// Mitsubishi GX Works2 project: BAJAJ-N5K-Q CONV-18.08.22_MOD2   PLC: Q03UDV

PROGRAM MAIN
0     END
END_PROGRAM

PROGRAM 1_ALARMS  // ALL
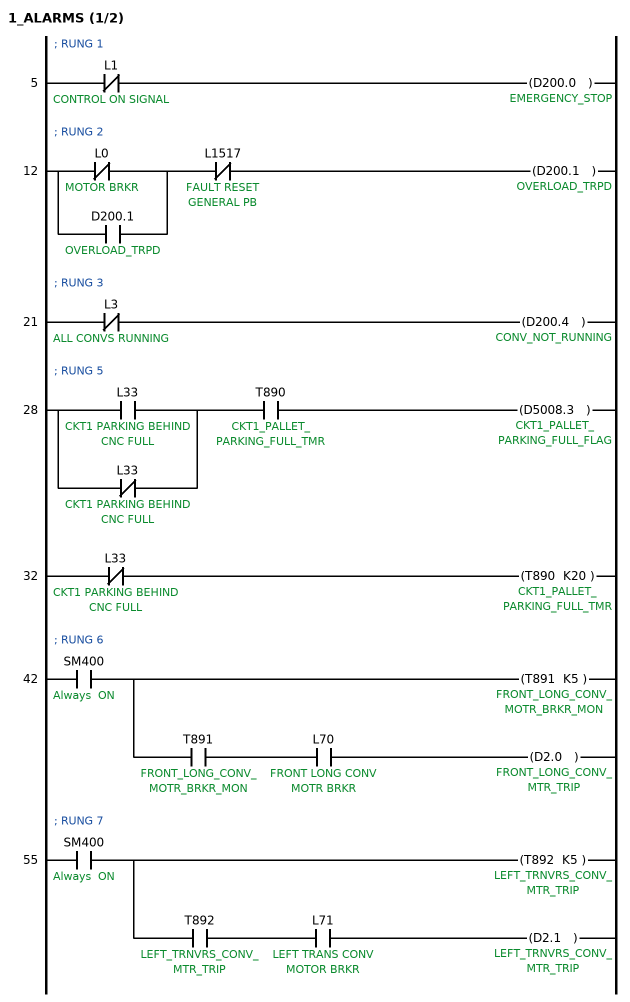
; RUNG 1
5     LDI     L1  ; CONTROL ON SIGNAL
      OUT     D200.0  ; EMERGENCY_STOP
; RUNG 2
12    LDI     L0  ; MOTOR BRKR
      OR      D200.1  ; OVERLOAD_TRPD
      ANI     L1517  ; FAULT RESET GENERAL PB
      OUT     D200.1  ; OVERLOAD_TRPD
; RUNG 3
21    LDI     L3  ; ALL CONVS RUNNING
      OUT     D200.4  ; CONV_NOT_RUNNING
; RUNG 5
28    LD      L33  ; CKT1 PARKING BEHIND CNC FULL
      ORI     L33  ; CKT1 PARKING BEHIND CNC FULL
      AND     T890  ; CKT1_PALLET_PARKING_FULL_TMR
      OUT     D5008.3  ; CKT1_PALLET_PARKING_FULL_FLAG
32    LDI     L33  ; CKT1 PARKING BEHIND CNC FULL
      OUT     T890 K20  ; CKT1_PALLET_PARKING_FULL_TMR
; RUNG 6
42    LD      SM400  ; Always  ON
      OUT     T891 K5  ; FRONT_LONG_CONV_MOTR_BRKR_MON
      AND     T891  ; FRONT_LONG_CONV_MOTR_BRKR_MON
      AND     L70  ; FRONT LONG CONV MOTR BRKR
      OUT     D2.0  ; FRONT_LONG_CONV_MTR_TRIP
; RUNG 7
55    LD      SM400  ; Always  ON
      OUT     T892 K5  ; LEFT_TRNVRS_CONV_MTR_TRIP
      AND     T892  ; LEFT_TRNVRS_CONV_MTR_TRIP
      AND     L71  ; LEFT TRANS CONV MOTOR BRKR
      OUT     D2.1  ; LEFT_TRNVRS_CONV_MTR_TRIP
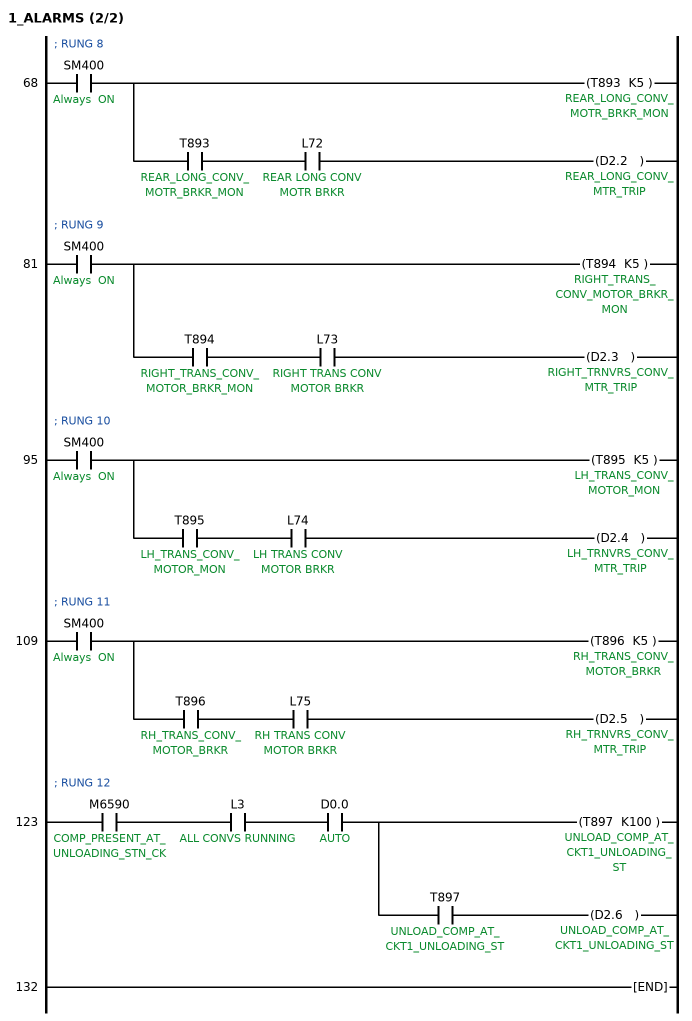
; RUNG 8
68    LD      SM400  ; Always  ON
      OUT     T893 K5  ; REAR_LONG_CONV_MOTR_BRKR_MON
      AND     T893  ; REAR_LONG_CONV_MOTR_BRKR_MON
      AND     L72  ; REAR LONG CONV MOTR BRKR
      OUT     D2.2  ; REAR_LONG_CONV_MTR_TRIP
; RUNG 9
81    LD      SM400  ; Always  ON
      OUT     T894 K5  ; RIGHT_TRANS_CONV_MOTOR_BRKR_MON
      AND     T894  ; RIGHT_TRANS_CONV_MOTOR_BRKR_MON
      AND     L73  ; RIGHT TRANS CONV MOTOR BRKR
      OUT     D2.3  ; RIGHT_TRNVRS_CONV_MTR_TRIP
; RUNG 10
95    LD      SM400  ; Always  ON
      OUT     T895 K5  ; LH_TRANS_CONV_MOTOR_MON
      AND     T895  ; LH_TRANS_CONV_MOTOR_MON
      AND     L74  ; LH TRANS CONV MOTOR BRKR
      OUT     D2.4  ; LH_TRNVRS_CONV_MTR_TRIP
; RUNG 11
109   LD      SM400  ; Always  ON
      OUT     T896 K5  ; RH_TRANS_CONV_MOTOR_BRKR
      AND     T896  ; RH_TRANS_CONV_MOTOR_BRKR
      AND     L75  ; RH TRANS CONV MOTOR BRKR
      OUT     D2.5  ; RH_TRNVRS_CONV_MTR_TRIP
; RUNG 12
123   LD      M6590  ; COMP_PRESENT_AT_UNLOADING_STN_CK
      AND     L3  ; ALL CONVS RUNNING
      AND     D0.0  ; AUTO
      OUT     T897 K100  ; UNLOAD_COMP_AT_CKT1_UNLOADING_ST
      AND     T897  ; UNLOAD_COMP_AT_CKT1_UNLOADING_ST
      OUT     D2.6  ; UNLOAD_COMP_AT_CKT1_UNLOADING_ST
132   END
END_PROGRAM

PROGRAM 2_AUTO  // UNLOADER
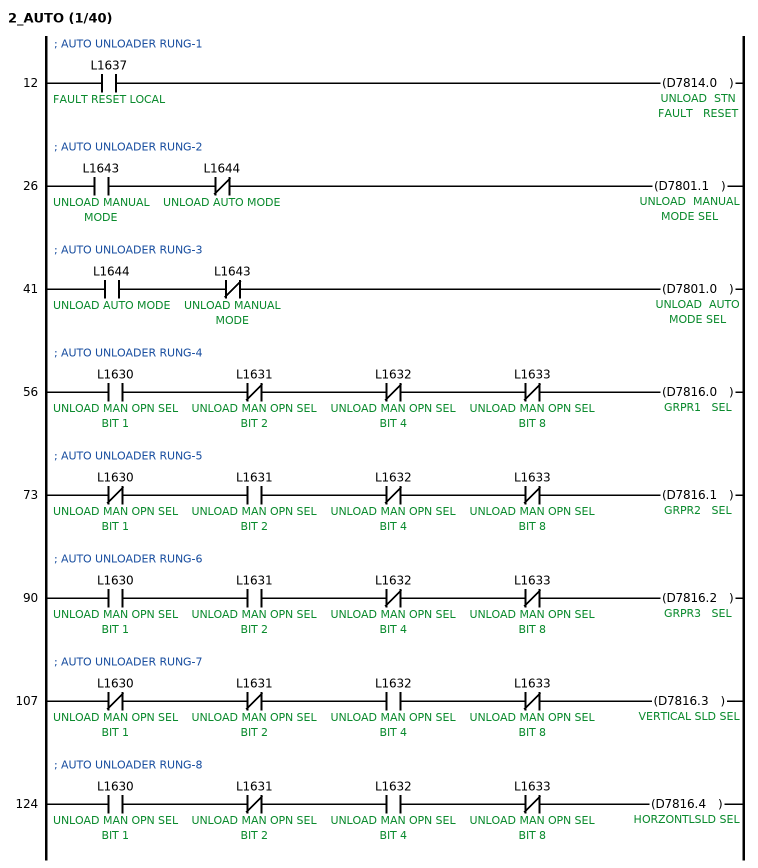
; AUTO UNLOADER RUNG-1
12    LD      L1637  ; FAULT RESET LOCAL
      OUT     D7814.0  ; UNLOAD  STN     FAULT   RESET
; AUTO UNLOADER RUNG-2
26    LD      L1643  ; UNLOAD MANUAL MODE
      ANI     L1644  ; UNLOAD AUTO MODE
      OUT     D7801.1  ; UNLOAD  MANUAL  MODE SEL
; AUTO UNLOADER RUNG-3
41    LD      L1644  ; UNLOAD AUTO MODE
      ANI     L1643  ; UNLOAD MANUAL MODE
      OUT     D7801.0  ; UNLOAD  AUTO    MODE SEL
; AUTO UNLOADER RUNG-4
56    LD      L1630  ; UNLOAD MAN OPN SEL BIT 1
      ANI     L1631  ; UNLOAD MAN OPN SEL BIT 2
      ANI     L1632  ; UNLOAD MAN OPN SEL BIT 4
      ANI     L1633  ; UNLOAD MAN OPN SEL BIT 8
      OUT     D7816.0  ; GRPR1   SEL
; AUTO UNLOADER RUNG-5
73    LDI     L1630  ; UNLOAD MAN OPN SEL BIT 1
      AND     L1631  ; UNLOAD MAN OPN SEL BIT 2
      ANI     L1632  ; UNLOAD MAN OPN SEL BIT 4
      ANI     L1633  ; UNLOAD MAN OPN SEL BIT 8
      OUT     D7816.1  ; GRPR2   SEL
; AUTO UNLOADER RUNG-6
90    LD      L1630  ; UNLOAD MAN OPN SEL BIT 1
      AND     L1631  ; UNLOAD MAN OPN SEL BIT 2
      ANI     L1632  ; UNLOAD MAN OPN SEL BIT 4
      ANI     L1633  ; UNLOAD MAN OPN SEL BIT 8
      OUT     D7816.2  ; GRPR3   SEL
; AUTO UNLOADER RUNG-7
107   LDI     L1630  ; UNLOAD MAN OPN SEL BIT 1
      ANI     L1631  ; UNLOAD MAN OPN SEL BIT 2
      AND     L1632  ; UNLOAD MAN OPN SEL BIT 4
      ANI     L1633  ; UNLOAD MAN OPN SEL BIT 8
      OUT     D7816.3  ; VERTICAL SLD SEL
; AUTO UNLOADER RUNG-8
124   LD      L1630  ; UNLOAD MAN OPN SEL BIT 1
      ANI     L1631  ; UNLOAD MAN OPN SEL BIT 2
      AND     L1632  ; UNLOAD MAN OPN SEL BIT 4
      ANI     L1633  ; UNLOAD MAN OPN SEL BIT 8
      OUT     D7816.4  ; HORZONTLSLD SEL
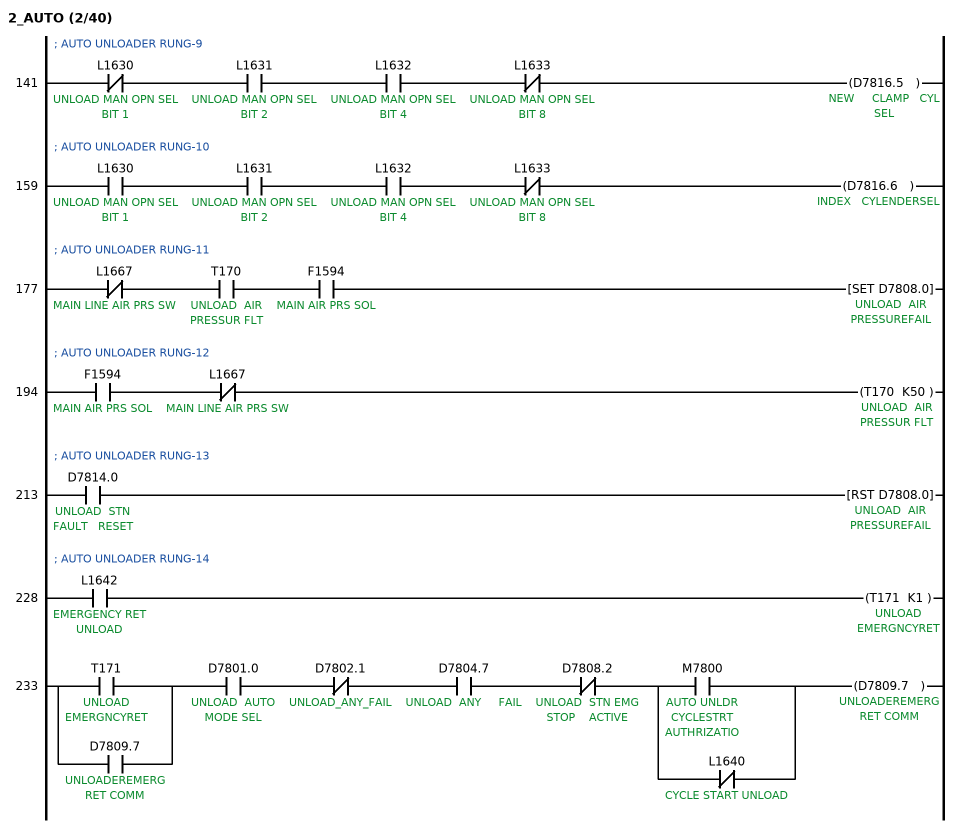
; AUTO UNLOADER RUNG-9
141   LDI     L1630  ; UNLOAD MAN OPN SEL BIT 1
      AND     L1631  ; UNLOAD MAN OPN SEL BIT 2
      AND     L1632  ; UNLOAD MAN OPN SEL BIT 4
      ANI     L1633  ; UNLOAD MAN OPN SEL BIT 8
      OUT     D7816.5  ; NEW     CLAMP   CYL SEL
; AUTO UNLOADER RUNG-10
159   LD      L1630  ; UNLOAD MAN OPN SEL BIT 1
      AND     L1631  ; UNLOAD MAN OPN SEL BIT 2
      AND     L1632  ; UNLOAD MAN OPN SEL BIT 4
      ANI     L1633  ; UNLOAD MAN OPN SEL BIT 8
      OUT     D7816.6  ; INDEX   CYLENDERSEL
; AUTO UNLOADER RUNG-11
177   LDI     L1667  ; MAIN LINE AIR PRS SW
      AND     T170  ; UNLOAD  AIR     PRESSUR FLT
      AND     F1594  ; MAIN AIR PRS SOL
      SET     D7808.0  ; UNLOAD  AIR     PRESSUREFAIL
; AUTO UNLOADER RUNG-12
194   LD      F1594  ; MAIN AIR PRS SOL
      ANI     L1667  ; MAIN LINE AIR PRS SW
      OUT     T170 K50  ; UNLOAD  AIR     PRESSUR FLT
; AUTO UNLOADER RUNG-13
213   LD      D7814.0  ; UNLOAD  STN     FAULT   RESET
      RST     D7808.0  ; UNLOAD  AIR     PRESSUREFAIL
; AUTO UNLOADER RUNG-14
228   LD      L1642  ; EMERGENCY RET UNLOAD
      OUT     T171 K1  ; UNLOAD  EMERGNCYRET
233   LD      T171  ; UNLOAD  EMERGNCYRET
      OR      D7809.7  ; UNLOADEREMERG   RET COMM
      AND     D7801.0  ; UNLOAD  AUTO    MODE SEL
      ANI     D7802.1  ; UNLOAD_ANY_FAIL
      AND     D7804.7  ; UNLOAD  ANY     FAIL
      ANI     D7808.2  ; UNLOAD  STN EMG STOP    ACTIVE
      LD      M7800  ; AUTO UNLDR CYCLESTRT AUTHRIZATIO
      ORI     L1640  ; CYCLE START UNLOAD
      ANB
      OUT     D7809.7  ; UNLOADEREMERG   RET COMM
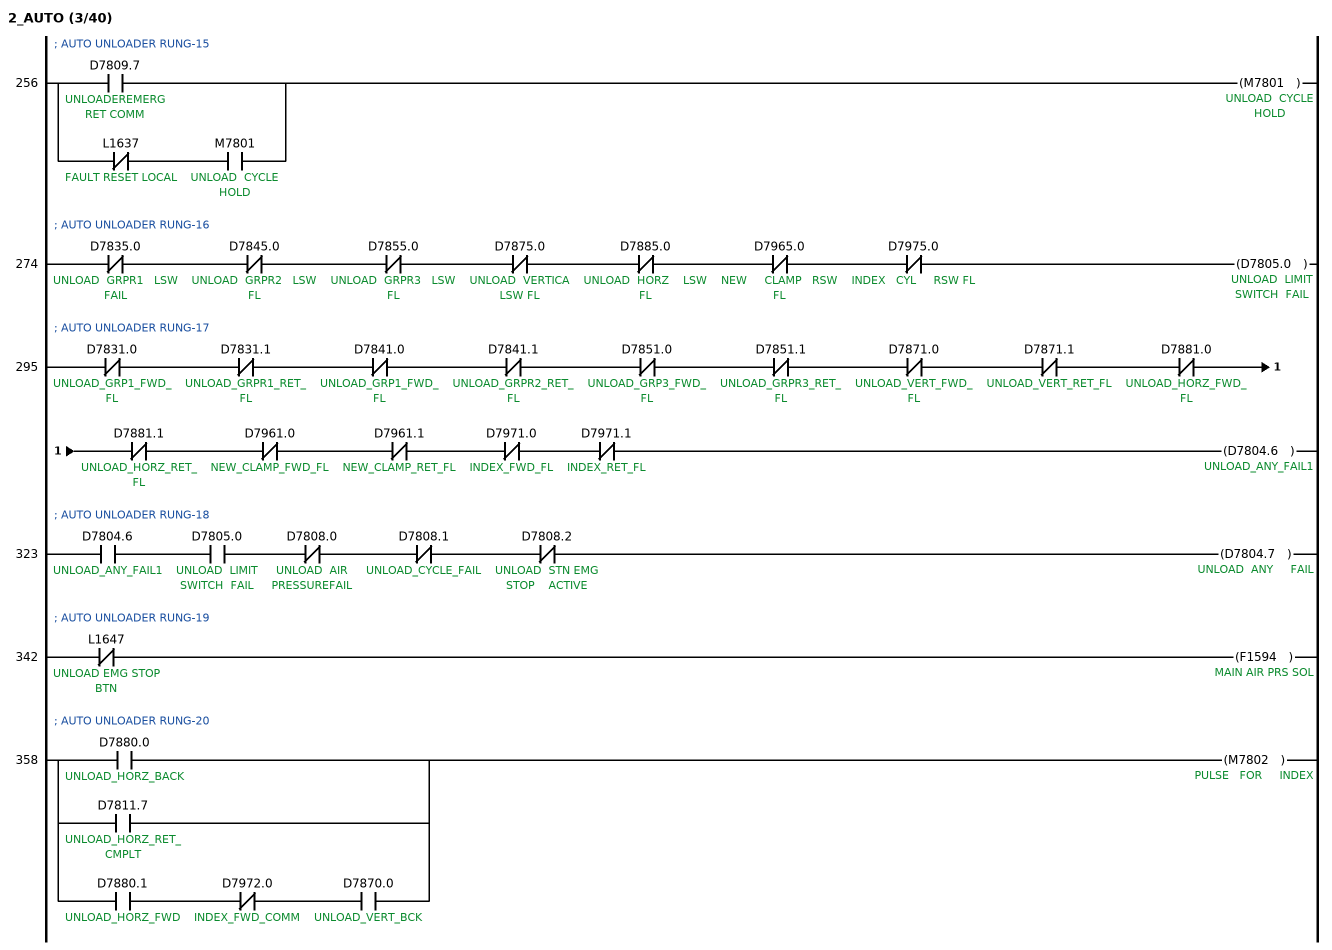
; AUTO UNLOADER RUNG-15
256   LD      D7809.7  ; UNLOADEREMERG   RET COMM
      LDI     L1637  ; FAULT RESET LOCAL
      AND     M7801  ; UNLOAD  CYCLE   HOLD
      ORB
      OUT     M7801  ; UNLOAD  CYCLE   HOLD
; AUTO UNLOADER RUNG-16
274   LDI     D7835.0  ; UNLOAD  GRPR1   LSW FAIL
      ANI     D7845.0  ; UNLOAD  GRPR2   LSW FL
      ANI     D7855.0  ; UNLOAD  GRPR3   LSW FL
      ANI     D7875.0  ; UNLOAD  VERTICA LSW FL
      ANI     D7885.0  ; UNLOAD  HORZ    LSW FL
      ANI     D7965.0  ; NEW     CLAMP   RSW FL
      ANI     D7975.0  ; INDEX   CYL     RSW FL
      OUT     D7805.0  ; UNLOAD  LIMIT   SWITCH  FAIL
; AUTO UNLOADER RUNG-17
295   LDI     D7831.0  ; UNLOAD_GRP1_FWD_FL
      ANI     D7831.1  ; UNLOAD_GRPR1_RET_FL
      ANI     D7841.0  ; UNLOAD_GRP1_FWD_FL
      ANI     D7841.1  ; UNLOAD_GRPR2_RET_FL
      ANI     D7851.0  ; UNLOAD_GRP3_FWD_FL
      ANI     D7851.1  ; UNLOAD_GRPR3_RET_FL
      ANI     D7871.0  ; UNLOAD_VERT_FWD_FL
      ANI     D7871.1  ; UNLOAD_VERT_RET_FL
      ANI     D7881.0  ; UNLOAD_HORZ_FWD_FL
      ANI     D7881.1  ; UNLOAD_HORZ_RET_FL
      ANI     D7961.0  ; NEW_CLAMP_FWD_FL
      ANI     D7961.1  ; NEW_CLAMP_RET_FL
      ANI     D7971.0  ; INDEX_FWD_FL
      ANI     D7971.1  ; INDEX_RET_FL
      OUT     D7804.6  ; UNLOAD_ANY_FAIL1
; AUTO UNLOADER RUNG-18
323   LD      D7804.6  ; UNLOAD_ANY_FAIL1
      AND     D7805.0  ; UNLOAD  LIMIT   SWITCH  FAIL
      ANI     D7808.0  ; UNLOAD  AIR     PRESSUREFAIL
      ANI     D7808.1  ; UNLOAD_CYCLE_FAIL
      ANI     D7808.2  ; UNLOAD  STN EMG STOP    ACTIVE
      OUT     D7804.7  ; UNLOAD  ANY     FAIL
; AUTO UNLOADER RUNG-19
342   LDI     L1647  ; UNLOAD EMG STOP BTN
      OUT     F1594  ; MAIN AIR PRS SOL
; AUTO UNLOADER RUNG-20
358   LD      D7880.0  ; UNLOAD_HORZ_BACK
      OR      D7811.7  ; UNLOAD_HORZ_RET_CMPLT
      LD      D7880.1  ; UNLOAD_HORZ_FWD
      ANI     D7972.0  ; INDEX_FWD_COMM
      AND     D7870.0  ; UNLOAD_VERT_BCK
      ORB
      OUT     M7802  ; PULSE   FOR     INDEX
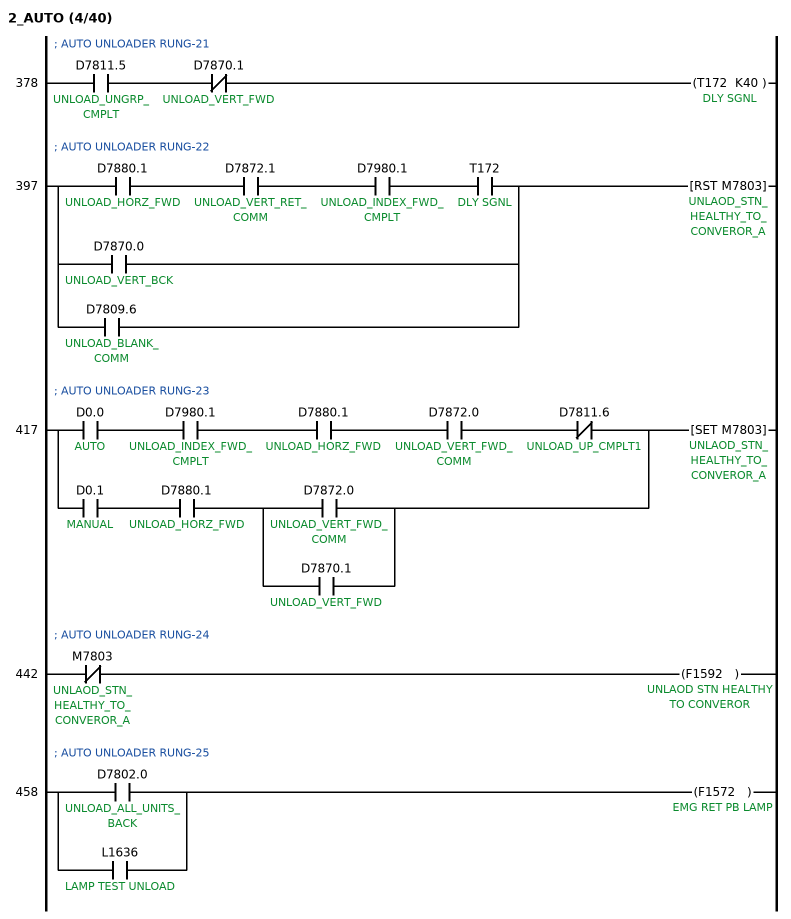
; AUTO UNLOADER RUNG-21
378   LD      D7811.5  ; UNLOAD_UNGRP_CMPLT
      ANI     D7870.1  ; UNLOAD_VERT_FWD
      OUT     T172 K40  ; DLY SGNL
; AUTO UNLOADER RUNG-22
397   LD      D7880.1  ; UNLOAD_HORZ_FWD
      AND     D7872.1  ; UNLOAD_VERT_RET_COMM
      AND     D7980.1  ; UNLOAD_INDEX_FWD_CMPLT
      AND     T172  ; DLY SGNL
      OR      D7870.0  ; UNLOAD_VERT_BCK
      OR      D7809.6  ; UNLOAD_BLANK_COMM
      RST     M7803  ; UNLAOD_STN_HEALTHY_TO_CONVEROR_A
; AUTO UNLOADER RUNG-23
417   LD      D0.0  ; AUTO
      AND     D7980.1  ; UNLOAD_INDEX_FWD_CMPLT
      AND     D7880.1  ; UNLOAD_HORZ_FWD
      AND     D7872.0  ; UNLOAD_VERT_FWD_COMM
      ANI     D7811.6  ; UNLOAD_UP_CMPLT1
      LD      D0.1  ; MANUAL
      AND     D7880.1  ; UNLOAD_HORZ_FWD
      LD      D7872.0  ; UNLOAD_VERT_FWD_COMM
      OR      D7870.1  ; UNLOAD_VERT_FWD
      ANB
      ORB
      SET     M7803  ; UNLAOD_STN_HEALTHY_TO_CONVEROR_A
; AUTO UNLOADER RUNG-24
442   LDI     M7803  ; UNLAOD_STN_HEALTHY_TO_CONVEROR_A
      OUT     F1592  ; UNLAOD STN HEALTHY TO CONVEROR
; AUTO UNLOADER RUNG-25
458   LD      D7802.0  ; UNLOAD_ALL_UNITS_BACK
      OR      L1636  ; LAMP TEST UNLOAD
      OUT     F1572  ; EMG RET PB LAMP
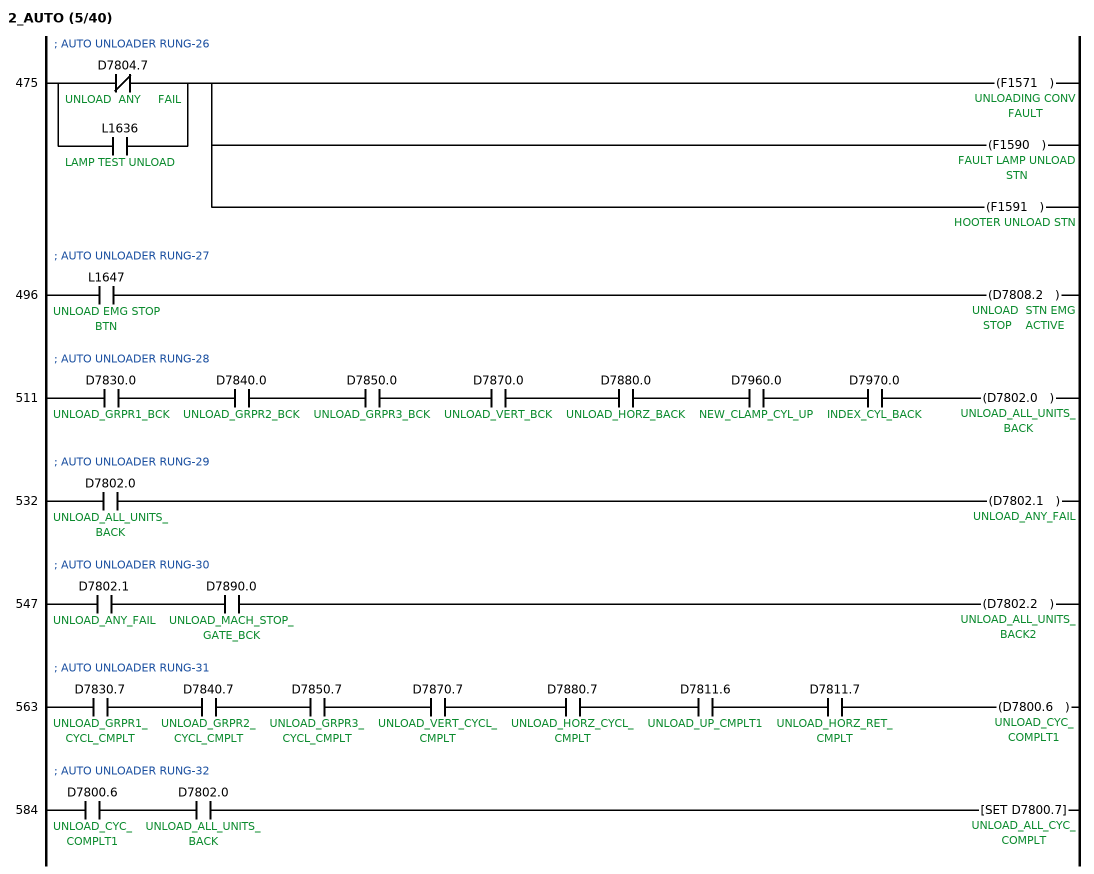
; AUTO UNLOADER RUNG-26
475   LDI     D7804.7  ; UNLOAD  ANY     FAIL
      OR      L1636  ; LAMP TEST UNLOAD
      OUT     F1571  ; UNLOADING CONV FAULT
      OUT     F1590  ; FAULT LAMP UNLOAD STN
      OUT     F1591  ; HOOTER UNLOAD STN
; AUTO UNLOADER RUNG-27
496   LD      L1647  ; UNLOAD EMG STOP BTN
      OUT     D7808.2  ; UNLOAD  STN EMG STOP    ACTIVE
; AUTO UNLOADER RUNG-28
511   LD      D7830.0  ; UNLOAD_GRPR1_BCK
      AND     D7840.0  ; UNLOAD_GRPR2_BCK
      AND     D7850.0  ; UNLOAD_GRPR3_BCK
      AND     D7870.0  ; UNLOAD_VERT_BCK
      AND     D7880.0  ; UNLOAD_HORZ_BACK
      AND     D7960.0  ; NEW_CLAMP_CYL_UP
      AND     D7970.0  ; INDEX_CYL_BACK
      OUT     D7802.0  ; UNLOAD_ALL_UNITS_BACK
; AUTO UNLOADER RUNG-29
532   LD      D7802.0  ; UNLOAD_ALL_UNITS_BACK
      OUT     D7802.1  ; UNLOAD_ANY_FAIL
; AUTO UNLOADER RUNG-30
547   LD      D7802.1  ; UNLOAD_ANY_FAIL
      AND     D7890.0  ; UNLOAD_MACH_STOP_GATE_BCK
      OUT     D7802.2  ; UNLOAD_ALL_UNITS_BACK2
; AUTO UNLOADER RUNG-31
563   LD      D7830.7  ; UNLOAD_GRPR1_CYCL_CMPLT
      AND     D7840.7  ; UNLOAD_GRPR2_CYCL_CMPLT
      AND     D7850.7  ; UNLOAD_GRPR3_CYCL_CMPLT
      AND     D7870.7  ; UNLOAD_VERT_CYCL_CMPLT
      AND     D7880.7  ; UNLOAD_HORZ_CYCL_CMPLT
      AND     D7811.6  ; UNLOAD_UP_CMPLT1
      AND     D7811.7  ; UNLOAD_HORZ_RET_CMPLT
      OUT     D7800.6  ; UNLOAD_CYC_COMPLT1
; AUTO UNLOADER RUNG-32
584   LD      D7800.6  ; UNLOAD_CYC_COMPLT1
      AND     D7802.0  ; UNLOAD_ALL_UNITS_BACK
      SET     D7800.7  ; UNLOAD_ALL_CYC_COMPLT
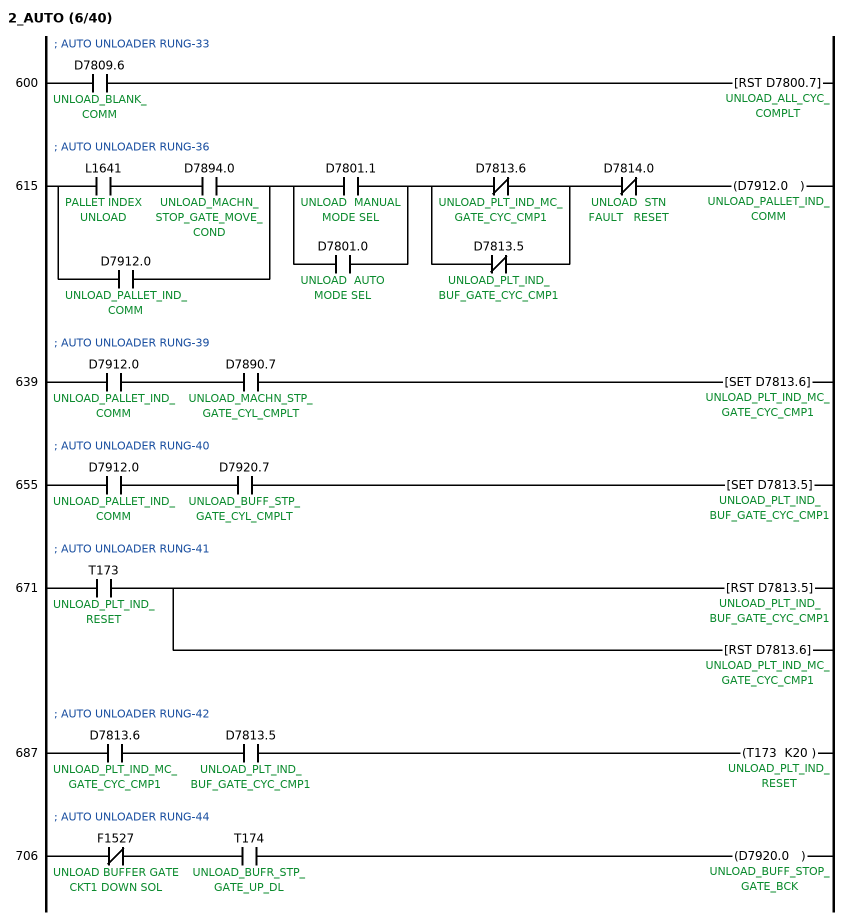
; AUTO UNLOADER RUNG-33
600   LD      D7809.6  ; UNLOAD_BLANK_COMM
      RST     D7800.7  ; UNLOAD_ALL_CYC_COMPLT
; AUTO UNLOADER RUNG-36
615   LD      L1641  ; PALLET INDEX UNLOAD
      AND     D7894.0  ; UNLOAD_MACHN_STOP_GATE_MOVE_COND
      OR      D7912.0  ; UNLOAD_PALLET_IND_COMM
      LD      D7801.1  ; UNLOAD  MANUAL  MODE SEL
      OR      D7801.0  ; UNLOAD  AUTO    MODE SEL
      ANB
      LDI     D7813.6  ; UNLOAD_PLT_IND_MC_GATE_CYC_CMP1
      ORI     D7813.5  ; UNLOAD_PLT_IND_BUF_GATE_CYC_CMP1
      ANB
      ANI     D7814.0  ; UNLOAD  STN     FAULT   RESET
      OUT     D7912.0  ; UNLOAD_PALLET_IND_COMM
; AUTO UNLOADER RUNG-39
639   LD      D7912.0  ; UNLOAD_PALLET_IND_COMM
      AND     D7890.7  ; UNLOAD_MACHN_STP_GATE_CYL_CMPLT
      SET     D7813.6  ; UNLOAD_PLT_IND_MC_GATE_CYC_CMP1
; AUTO UNLOADER RUNG-40
655   LD      D7912.0  ; UNLOAD_PALLET_IND_COMM
      AND     D7920.7  ; UNLOAD_BUFF_STP_GATE_CYL_CMPLT
      SET     D7813.5  ; UNLOAD_PLT_IND_BUF_GATE_CYC_CMP1
; AUTO UNLOADER RUNG-41
671   LD      T173  ; UNLOAD_PLT_IND_RESET
      RST     D7813.5  ; UNLOAD_PLT_IND_BUF_GATE_CYC_CMP1
      RST     D7813.6  ; UNLOAD_PLT_IND_MC_GATE_CYC_CMP1
; AUTO UNLOADER RUNG-42
687   LD      D7813.6  ; UNLOAD_PLT_IND_MC_GATE_CYC_CMP1
      AND     D7813.5  ; UNLOAD_PLT_IND_BUF_GATE_CYC_CMP1
      OUT     T173 K20  ; UNLOAD_PLT_IND_RESET
; AUTO UNLOADER RUNG-44
706   LDI     F1527  ; UNLOAD BUFFER GATE CKT1 DOWN SOL
      AND     T174  ; UNLOAD_BUFR_STP_GATE_UP_DL
      OUT     D7920.0  ; UNLOAD_BUFF_STOP_GATE_BCK
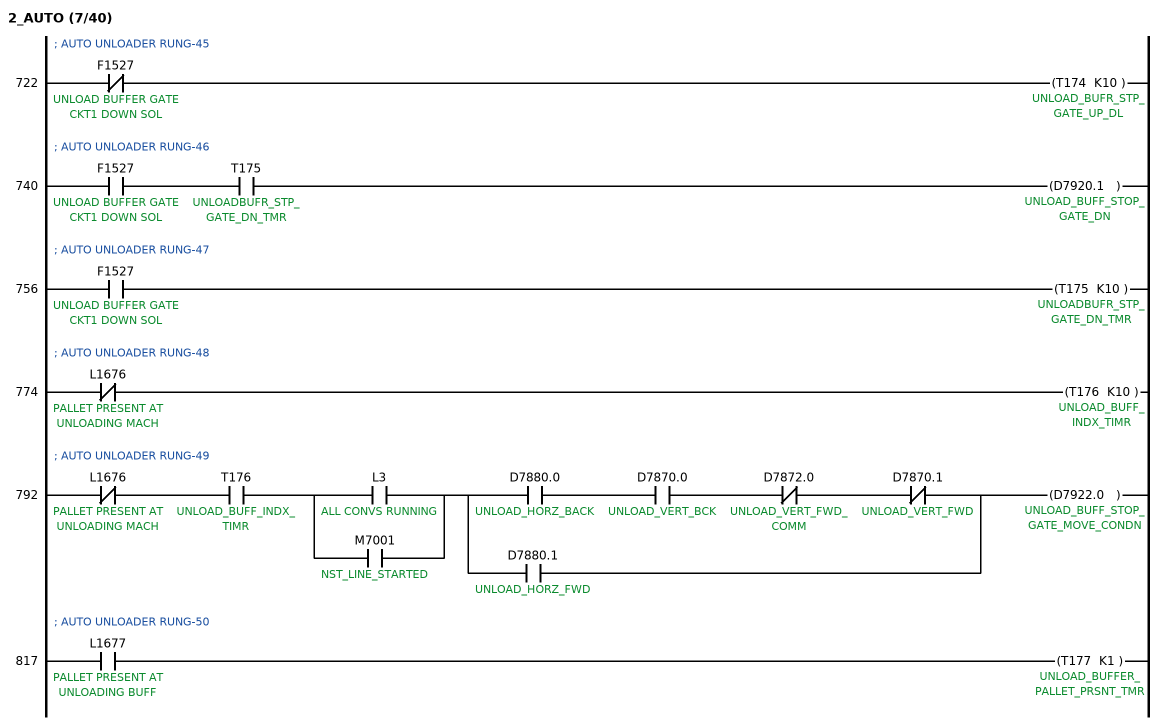
; AUTO UNLOADER RUNG-45
722   LDI     F1527  ; UNLOAD BUFFER GATE CKT1 DOWN SOL
      OUT     T174 K10  ; UNLOAD_BUFR_STP_GATE_UP_DL
; AUTO UNLOADER RUNG-46
740   LD      F1527  ; UNLOAD BUFFER GATE CKT1 DOWN SOL
      AND     T175  ; UNLOADBUFR_STP_GATE_DN_TMR
      OUT     D7920.1  ; UNLOAD_BUFF_STOP_GATE_DN
; AUTO UNLOADER RUNG-47
756   LD      F1527  ; UNLOAD BUFFER GATE CKT1 DOWN SOL
      OUT     T175 K10  ; UNLOADBUFR_STP_GATE_DN_TMR
; AUTO UNLOADER RUNG-48
774   LDI     L1676  ; PALLET PRESENT AT UNLOADING MACH
      OUT     T176 K10  ; UNLOAD_BUFF_INDX_TIMR
; AUTO UNLOADER RUNG-49
792   LDI     L1676  ; PALLET PRESENT AT UNLOADING MACH
      AND     T176  ; UNLOAD_BUFF_INDX_TIMR
      LD      L3  ; ALL CONVS RUNNING
      OR      M7001  ; NST_LINE_STARTED
      ANB
      LD      D7880.0  ; UNLOAD_HORZ_BACK
      AND     D7870.0  ; UNLOAD_VERT_BCK
      ANI     D7872.0  ; UNLOAD_VERT_FWD_COMM
      ANI     D7870.1  ; UNLOAD_VERT_FWD
      OR      D7880.1  ; UNLOAD_HORZ_FWD
      ANB
      OUT     D7922.0  ; UNLOAD_BUFF_STOP_GATE_MOVE_CONDN
; AUTO UNLOADER RUNG-50
817   LD      L1677  ; PALLET PRESENT AT UNLOADING BUFF
      OUT     T177 K1  ; UNLOAD_BUFFER_PALLET_PRSNT_TMR
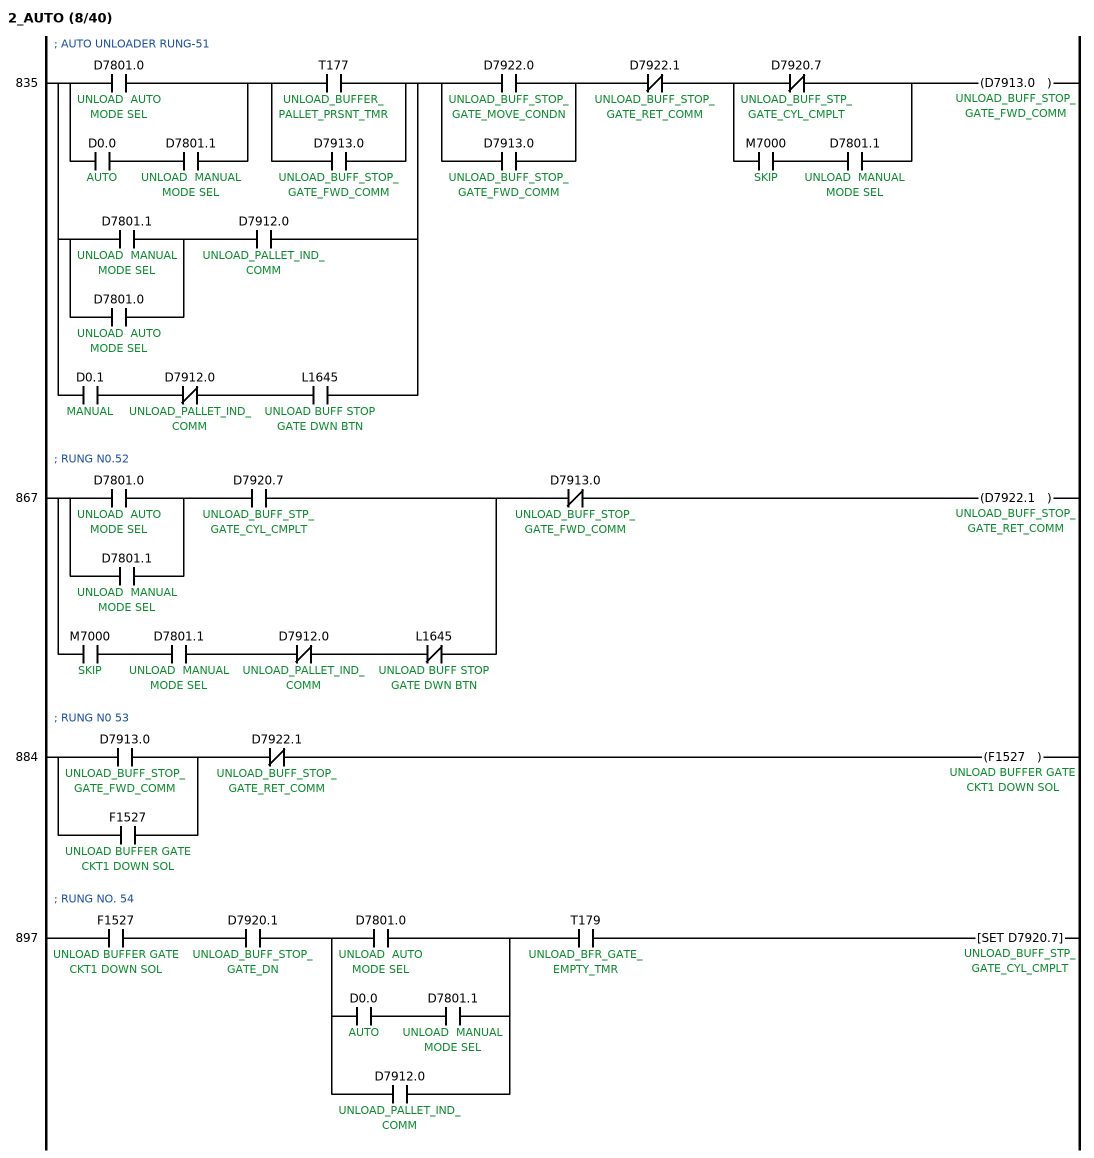
; AUTO UNLOADER RUNG-51
835   LD      D7801.0  ; UNLOAD  AUTO    MODE SEL
      LD      D0.0  ; AUTO
      AND     D7801.1  ; UNLOAD  MANUAL  MODE SEL
      ORB
      LD      T177  ; UNLOAD_BUFFER_PALLET_PRSNT_TMR
      OR      D7913.0  ; UNLOAD_BUFF_STOP_GATE_FWD_COMM
      ANB
      LD      D7801.1  ; UNLOAD  MANUAL  MODE SEL
      OR      D7801.0  ; UNLOAD  AUTO    MODE SEL
      AND     D7912.0  ; UNLOAD_PALLET_IND_COMM
      ORB
      LD      D0.1  ; MANUAL
      ANI     D7912.0  ; UNLOAD_PALLET_IND_COMM
      AND     L1645  ; UNLOAD BUFF STOP GATE DWN BTN
      ORB
      LD      D7922.0  ; UNLOAD_BUFF_STOP_GATE_MOVE_CONDN
      OR      D7913.0  ; UNLOAD_BUFF_STOP_GATE_FWD_COMM
      ANB
      ANI     D7922.1  ; UNLOAD_BUFF_STOP_GATE_RET_COMM
      LDI     D7920.7  ; UNLOAD_BUFF_STP_GATE_CYL_CMPLT
      LD      M7000  ; SKIP
      AND     D7801.1  ; UNLOAD  MANUAL  MODE SEL
      ORB
      ANB
      OUT     D7913.0  ; UNLOAD_BUFF_STOP_GATE_FWD_COMM
; RUNG N0.52
867   LD      D7801.0  ; UNLOAD  AUTO    MODE SEL
      OR      D7801.1  ; UNLOAD  MANUAL  MODE SEL
      AND     D7920.7  ; UNLOAD_BUFF_STP_GATE_CYL_CMPLT
      LD      M7000  ; SKIP
      AND     D7801.1  ; UNLOAD  MANUAL  MODE SEL
      ANI     D7912.0  ; UNLOAD_PALLET_IND_COMM
      ANI     L1645  ; UNLOAD BUFF STOP GATE DWN BTN
      ORB
      ANI     D7913.0  ; UNLOAD_BUFF_STOP_GATE_FWD_COMM
      OUT     D7922.1  ; UNLOAD_BUFF_STOP_GATE_RET_COMM
; RUNG N0 53
884   LD      D7913.0  ; UNLOAD_BUFF_STOP_GATE_FWD_COMM
      OR      F1527  ; UNLOAD BUFFER GATE CKT1 DOWN SOL
      ANI     D7922.1  ; UNLOAD_BUFF_STOP_GATE_RET_COMM
      OUT     F1527  ; UNLOAD BUFFER GATE CKT1 DOWN SOL
; RUNG NO. 54
897   LD      F1527  ; UNLOAD BUFFER GATE CKT1 DOWN SOL
      AND     D7920.1  ; UNLOAD_BUFF_STOP_GATE_DN
      LD      D7801.0  ; UNLOAD  AUTO    MODE SEL
      LD      D0.0  ; AUTO
      AND     D7801.1  ; UNLOAD  MANUAL  MODE SEL
      ORB
      OR      D7912.0  ; UNLOAD_PALLET_IND_COMM
      ANB
      AND     T179  ; UNLOAD_BFR_GATE_EMPTY_TMR
      SET     D7920.7  ; UNLOAD_BUFF_STP_GATE_CYL_CMPLT
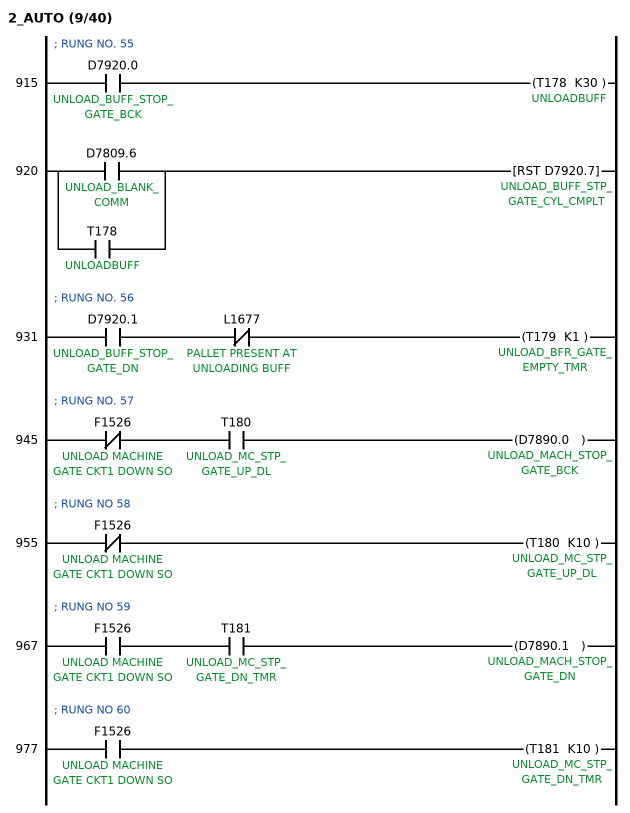
; RUNG NO. 55
915   LD      D7920.0  ; UNLOAD_BUFF_STOP_GATE_BCK
      OUT     T178 K30  ; UNLOADBUFF
920   LD      D7809.6  ; UNLOAD_BLANK_COMM
      OR      T178  ; UNLOADBUFF
      RST     D7920.7  ; UNLOAD_BUFF_STP_GATE_CYL_CMPLT
; RUNG NO. 56
931   LD      D7920.1  ; UNLOAD_BUFF_STOP_GATE_DN
      ANI     L1677  ; PALLET PRESENT AT UNLOADING BUFF
      OUT     T179 K1  ; UNLOAD_BFR_GATE_EMPTY_TMR
; RUNG NO. 57
945   LDI     F1526  ; UNLOAD MACHINE GATE CKT1 DOWN SO
      AND     T180  ; UNLOAD_MC_STP_GATE_UP_DL
      OUT     D7890.0  ; UNLOAD_MACH_STOP_GATE_BCK
; RUNG NO 58
955   LDI     F1526  ; UNLOAD MACHINE GATE CKT1 DOWN SO
      OUT     T180 K10  ; UNLOAD_MC_STP_GATE_UP_DL
; RUNG NO 59
967   LD      F1526  ; UNLOAD MACHINE GATE CKT1 DOWN SO
      AND     T181  ; UNLOAD_MC_STP_GATE_DN_TMR
      OUT     D7890.1  ; UNLOAD_MACH_STOP_GATE_DN
; RUNG NO 60
977   LD      F1526  ; UNLOAD MACHINE GATE CKT1 DOWN SO
      OUT     T181 K10  ; UNLOAD_MC_STP_GATE_DN_TMR
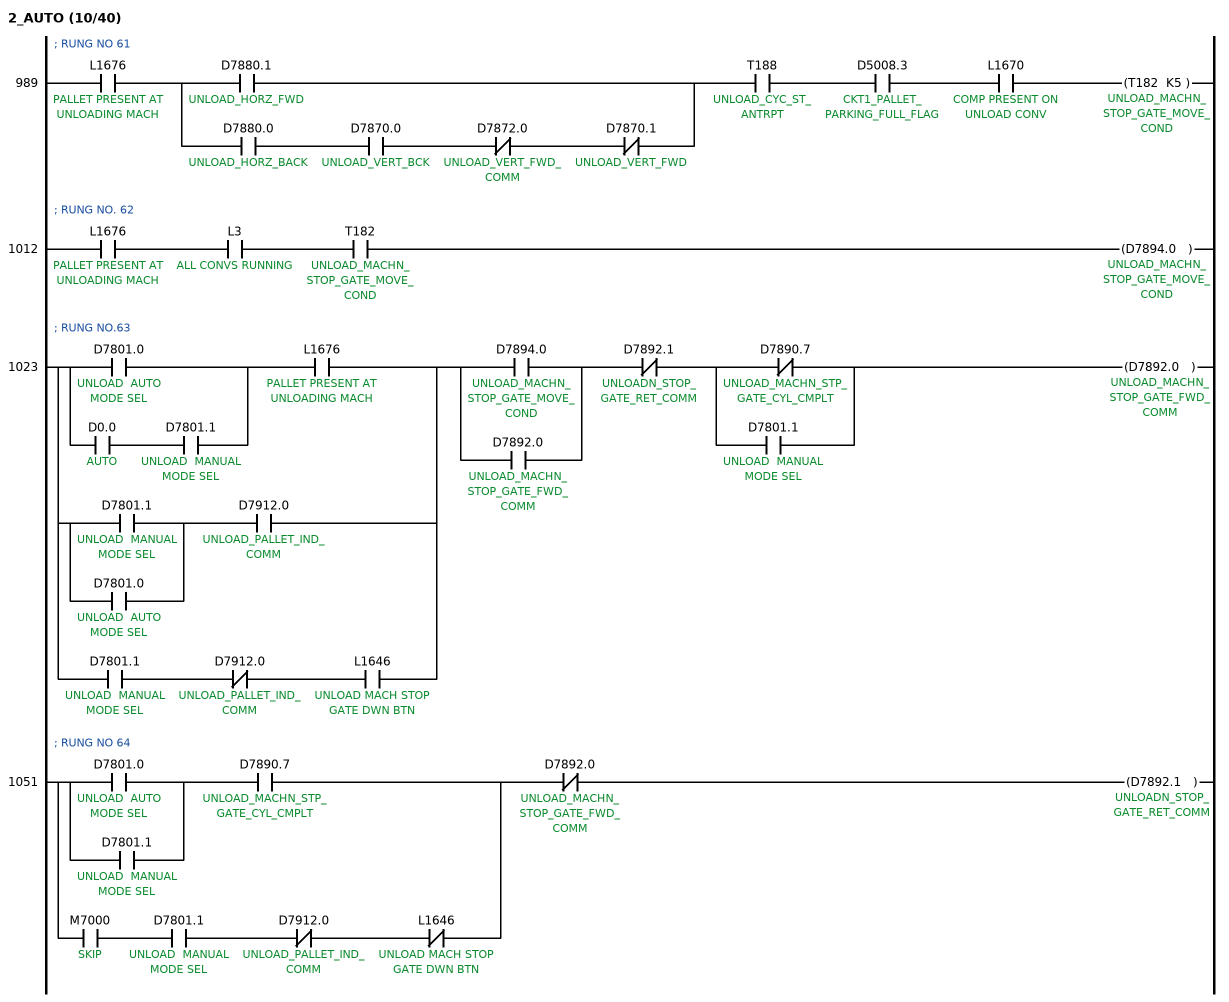
; RUNG NO 61
989   LD      L1676  ; PALLET PRESENT AT UNLOADING MACH
      LD      D7880.1  ; UNLOAD_HORZ_FWD
      LD      D7880.0  ; UNLOAD_HORZ_BACK
      AND     D7870.0  ; UNLOAD_VERT_BCK
      ANI     D7872.0  ; UNLOAD_VERT_FWD_COMM
      ANI     D7870.1  ; UNLOAD_VERT_FWD
      ORB
      ANB
      AND     T188  ; UNLOAD_CYC_ST_ANTRPT
      AND     D5008.3  ; CKT1_PALLET_PARKING_FULL_FLAG
      AND     L1670  ; COMP PRESENT ON UNLOAD CONV
      OUT     T182 K5  ; UNLOAD_MACHN_STOP_GATE_MOVE_COND
; RUNG NO. 62
1012  LD      L1676  ; PALLET PRESENT AT UNLOADING MACH
      AND     L3  ; ALL CONVS RUNNING
      AND     T182  ; UNLOAD_MACHN_STOP_GATE_MOVE_COND
      OUT     D7894.0  ; UNLOAD_MACHN_STOP_GATE_MOVE_COND
; RUNG NO.63
1023  LD      D7801.0  ; UNLOAD  AUTO    MODE SEL
      LD      D0.0  ; AUTO
      AND     D7801.1  ; UNLOAD  MANUAL  MODE SEL
      ORB
      AND     L1676  ; PALLET PRESENT AT UNLOADING MACH
      LD      D7801.1  ; UNLOAD  MANUAL  MODE SEL
      OR      D7801.0  ; UNLOAD  AUTO    MODE SEL
      AND     D7912.0  ; UNLOAD_PALLET_IND_COMM
      ORB
      LD      D7801.1  ; UNLOAD  MANUAL  MODE SEL
      ANI     D7912.0  ; UNLOAD_PALLET_IND_COMM
      AND     L1646  ; UNLOAD MACH STOP GATE DWN BTN
      ORB
      LD      D7894.0  ; UNLOAD_MACHN_STOP_GATE_MOVE_COND
      OR      D7892.0  ; UNLOAD_MACHN_STOP_GATE_FWD_COMM
      ANB
      ANI     D7892.1  ; UNLOADN_STOP_GATE_RET_COMM
      LDI     D7890.7  ; UNLOAD_MACHN_STP_GATE_CYL_CMPLT
      OR      D7801.1  ; UNLOAD  MANUAL  MODE SEL
      ANB
      OUT     D7892.0  ; UNLOAD_MACHN_STOP_GATE_FWD_COMM
; RUNG NO 64
1051  LD      D7801.0  ; UNLOAD  AUTO    MODE SEL
      OR      D7801.1  ; UNLOAD  MANUAL  MODE SEL
      AND     D7890.7  ; UNLOAD_MACHN_STP_GATE_CYL_CMPLT
      LD      M7000  ; SKIP
      AND     D7801.1  ; UNLOAD  MANUAL  MODE SEL
      ANI     D7912.0  ; UNLOAD_PALLET_IND_COMM
      ANI     L1646  ; UNLOAD MACH STOP GATE DWN BTN
      ORB
      ANI     D7892.0  ; UNLOAD_MACHN_STOP_GATE_FWD_COMM
      OUT     D7892.1  ; UNLOADN_STOP_GATE_RET_COMM
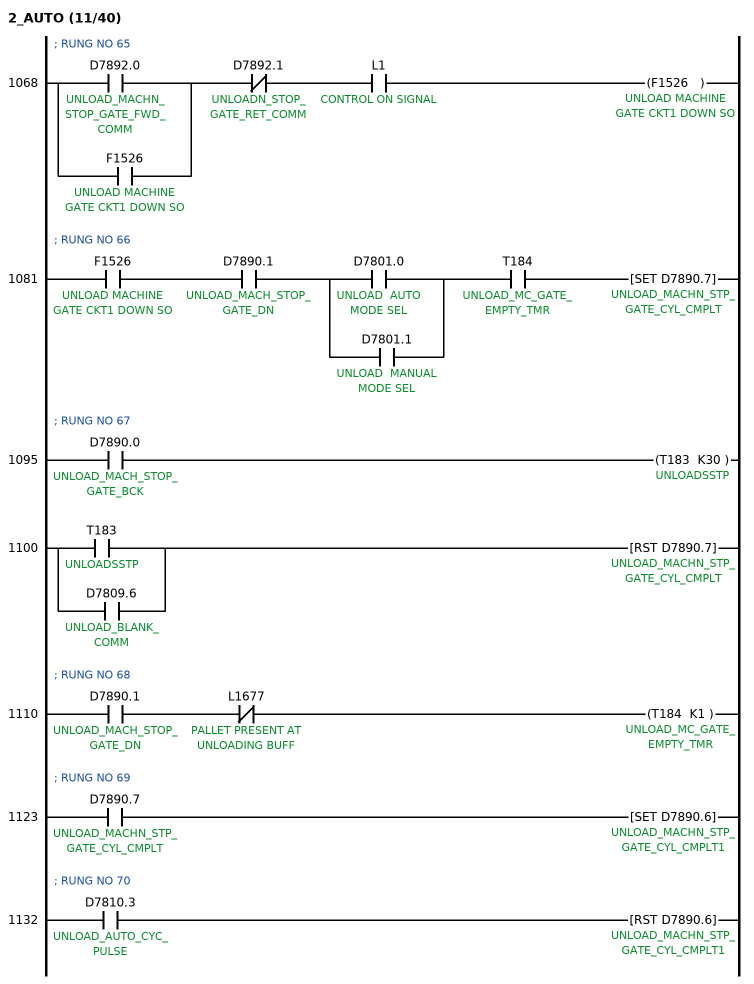
; RUNG NO 65
1068  LD      D7892.0  ; UNLOAD_MACHN_STOP_GATE_FWD_COMM
      OR      F1526  ; UNLOAD MACHINE GATE CKT1 DOWN SO
      ANI     D7892.1  ; UNLOADN_STOP_GATE_RET_COMM
      AND     L1  ; CONTROL ON SIGNAL
      OUT     F1526  ; UNLOAD MACHINE GATE CKT1 DOWN SO
; RUNG NO 66
1081  LD      F1526  ; UNLOAD MACHINE GATE CKT1 DOWN SO
      AND     D7890.1  ; UNLOAD_MACH_STOP_GATE_DN
      LD      D7801.0  ; UNLOAD  AUTO    MODE SEL
      OR      D7801.1  ; UNLOAD  MANUAL  MODE SEL
      ANB
      AND     T184  ; UNLOAD_MC_GATE_EMPTY_TMR
      SET     D7890.7  ; UNLOAD_MACHN_STP_GATE_CYL_CMPLT
; RUNG NO 67
1095  LD      D7890.0  ; UNLOAD_MACH_STOP_GATE_BCK
      OUT     T183 K30  ; UNLOADSSTP
1100  LD      T183  ; UNLOADSSTP
      OR      D7809.6  ; UNLOAD_BLANK_COMM
      RST     D7890.7  ; UNLOAD_MACHN_STP_GATE_CYL_CMPLT
; RUNG NO 68
1110  LD      D7890.1  ; UNLOAD_MACH_STOP_GATE_DN
      ANI     L1677  ; PALLET PRESENT AT UNLOADING BUFF
      OUT     T184 K1  ; UNLOAD_MC_GATE_EMPTY_TMR
; RUNG NO 69
1123  LD      D7890.7  ; UNLOAD_MACHN_STP_GATE_CYL_CMPLT
      SET     D7890.6  ; UNLOAD_MACHN_STP_GATE_CYL_CMPLT1
; RUNG NO 70
1132  LD      D7810.3  ; UNLOAD_AUTO_CYC_PULSE
      RST     D7890.6  ; UNLOAD_MACHN_STP_GATE_CYL_CMPLT1
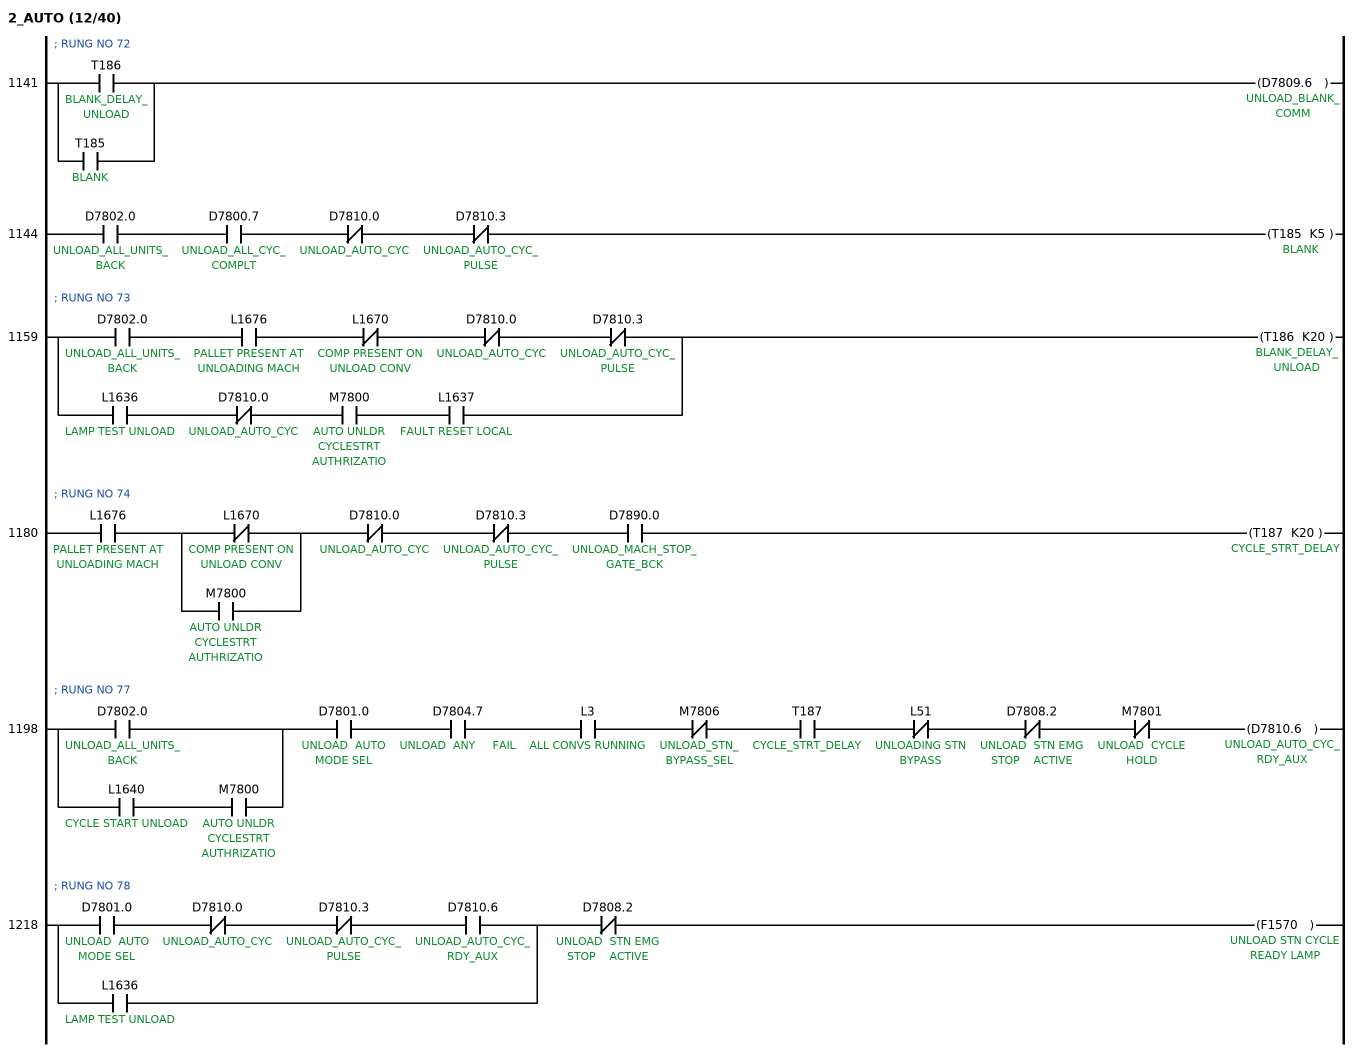
; RUNG NO 72
1141  LD      T186  ; BLANK_DELAY_UNLOAD
      OR      T185  ; BLANK
      OUT     D7809.6  ; UNLOAD_BLANK_COMM
1144  LD      D7802.0  ; UNLOAD_ALL_UNITS_BACK
      AND     D7800.7  ; UNLOAD_ALL_CYC_COMPLT
      ANI     D7810.0  ; UNLOAD_AUTO_CYC
      ANI     D7810.3  ; UNLOAD_AUTO_CYC_PULSE
      OUT     T185 K5  ; BLANK
; RUNG NO 73
1159  LD      D7802.0  ; UNLOAD_ALL_UNITS_BACK
      AND     L1676  ; PALLET PRESENT AT UNLOADING MACH
      ANI     L1670  ; COMP PRESENT ON UNLOAD CONV
      ANI     D7810.0  ; UNLOAD_AUTO_CYC
      ANI     D7810.3  ; UNLOAD_AUTO_CYC_PULSE
      LD      L1636  ; LAMP TEST UNLOAD
      ANI     D7810.0  ; UNLOAD_AUTO_CYC
      AND     M7800  ; AUTO UNLDR CYCLESTRT AUTHRIZATIO
      AND     L1637  ; FAULT RESET LOCAL
      ORB
      OUT     T186 K20  ; BLANK_DELAY_UNLOAD
; RUNG NO 74
1180  LD      L1676  ; PALLET PRESENT AT UNLOADING MACH
      LDI     L1670  ; COMP PRESENT ON UNLOAD CONV
      OR      M7800  ; AUTO UNLDR CYCLESTRT AUTHRIZATIO
      ANB
      ANI     D7810.0  ; UNLOAD_AUTO_CYC
      ANI     D7810.3  ; UNLOAD_AUTO_CYC_PULSE
      AND     D7890.0  ; UNLOAD_MACH_STOP_GATE_BCK
      OUT     T187 K20  ; CYCLE_STRT_DELAY
; RUNG NO 77
1198  LD      D7802.0  ; UNLOAD_ALL_UNITS_BACK
      LD      L1640  ; CYCLE START UNLOAD
      AND     M7800  ; AUTO UNLDR CYCLESTRT AUTHRIZATIO
      ORB
      AND     D7801.0  ; UNLOAD  AUTO    MODE SEL
      AND     D7804.7  ; UNLOAD  ANY     FAIL
      AND     L3  ; ALL CONVS RUNNING
      ANI     M7806  ; UNLOAD_STN_BYPASS_SEL
      AND     T187  ; CYCLE_STRT_DELAY
      ANI     L51  ; UNLOADING STN BYPASS
      ANI     D7808.2  ; UNLOAD  STN EMG STOP    ACTIVE
      ANI     M7801  ; UNLOAD  CYCLE   HOLD
      OUT     D7810.6  ; UNLOAD_AUTO_CYC_RDY_AUX
; RUNG NO 78
1218  LD      D7801.0  ; UNLOAD  AUTO    MODE SEL
      ANI     D7810.0  ; UNLOAD_AUTO_CYC
      ANI     D7810.3  ; UNLOAD_AUTO_CYC_PULSE
      AND     D7810.6  ; UNLOAD_AUTO_CYC_RDY_AUX
      OR      L1636  ; LAMP TEST UNLOAD
      ANI     D7808.2  ; UNLOAD  STN EMG STOP    ACTIVE
      OUT     F1570  ; UNLOAD STN CYCLE READY LAMP
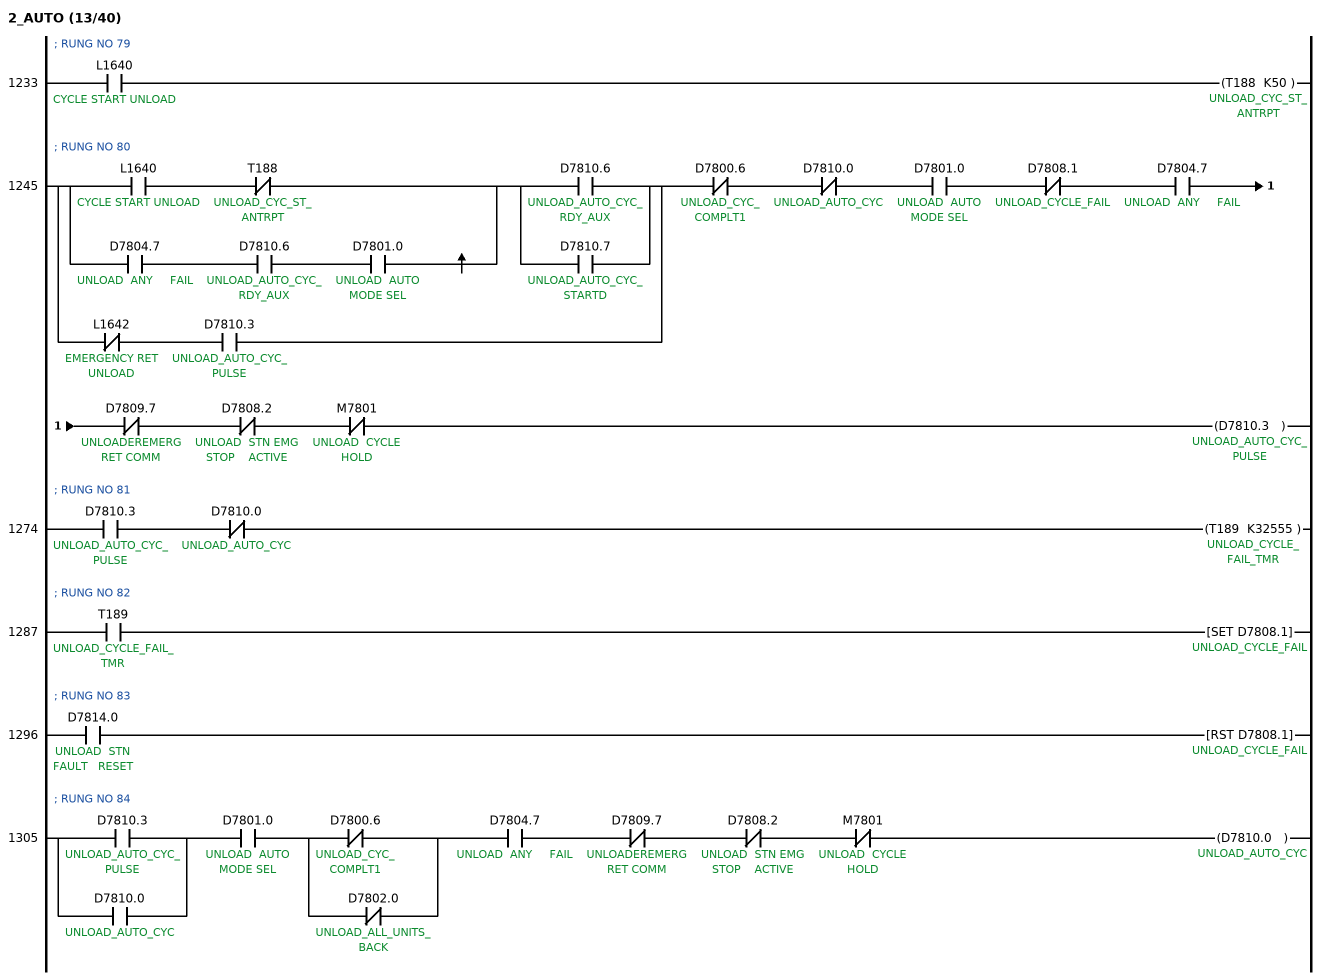
; RUNG NO 79
1233  LD      L1640  ; CYCLE START UNLOAD
      OUT     T188 K50  ; UNLOAD_CYC_ST_ANTRPT
; RUNG NO 80
1245  LD      L1640  ; CYCLE START UNLOAD
      ANI     T188  ; UNLOAD_CYC_ST_ANTRPT
      LD      D7804.7  ; UNLOAD  ANY     FAIL
      AND     D7810.6  ; UNLOAD_AUTO_CYC_RDY_AUX
      AND     D7801.0  ; UNLOAD  AUTO    MODE SEL
      MEP
      ORB
      LD      D7810.6  ; UNLOAD_AUTO_CYC_RDY_AUX
      OR      D7810.7  ; UNLOAD_AUTO_CYC_STARTD
      ANB
      LDI     L1642  ; EMERGENCY RET UNLOAD
      AND     D7810.3  ; UNLOAD_AUTO_CYC_PULSE
      ORB
      ANI     D7800.6  ; UNLOAD_CYC_COMPLT1
      ANI     D7810.0  ; UNLOAD_AUTO_CYC
      AND     D7801.0  ; UNLOAD  AUTO    MODE SEL
      ANI     D7808.1  ; UNLOAD_CYCLE_FAIL
      AND     D7804.7  ; UNLOAD  ANY     FAIL
      ANI     D7809.7  ; UNLOADEREMERG   RET COMM
      ANI     D7808.2  ; UNLOAD  STN EMG STOP    ACTIVE
      ANI     M7801  ; UNLOAD  CYCLE   HOLD
      OUT     D7810.3  ; UNLOAD_AUTO_CYC_PULSE
; RUNG NO 81
1274  LD      D7810.3  ; UNLOAD_AUTO_CYC_PULSE
      ANI     D7810.0  ; UNLOAD_AUTO_CYC
      OUT     T189 K32555  ; UNLOAD_CYCLE_FAIL_TMR
; RUNG NO 82
1287  LD      T189  ; UNLOAD_CYCLE_FAIL_TMR
      SET     D7808.1  ; UNLOAD_CYCLE_FAIL
; RUNG NO 83
1296  LD      D7814.0  ; UNLOAD  STN     FAULT   RESET
      RST     D7808.1  ; UNLOAD_CYCLE_FAIL
; RUNG NO 84
1305  LD      D7810.3  ; UNLOAD_AUTO_CYC_PULSE
      OR      D7810.0  ; UNLOAD_AUTO_CYC
      AND     D7801.0  ; UNLOAD  AUTO    MODE SEL
      LDI     D7800.6  ; UNLOAD_CYC_COMPLT1
      ORI     D7802.0  ; UNLOAD_ALL_UNITS_BACK
      ANB
      AND     D7804.7  ; UNLOAD  ANY     FAIL
      ANI     D7809.7  ; UNLOADEREMERG   RET COMM
      ANI     D7808.2  ; UNLOAD  STN EMG STOP    ACTIVE
      ANI     M7801  ; UNLOAD  CYCLE   HOLD
      OUT     D7810.0  ; UNLOAD_AUTO_CYC
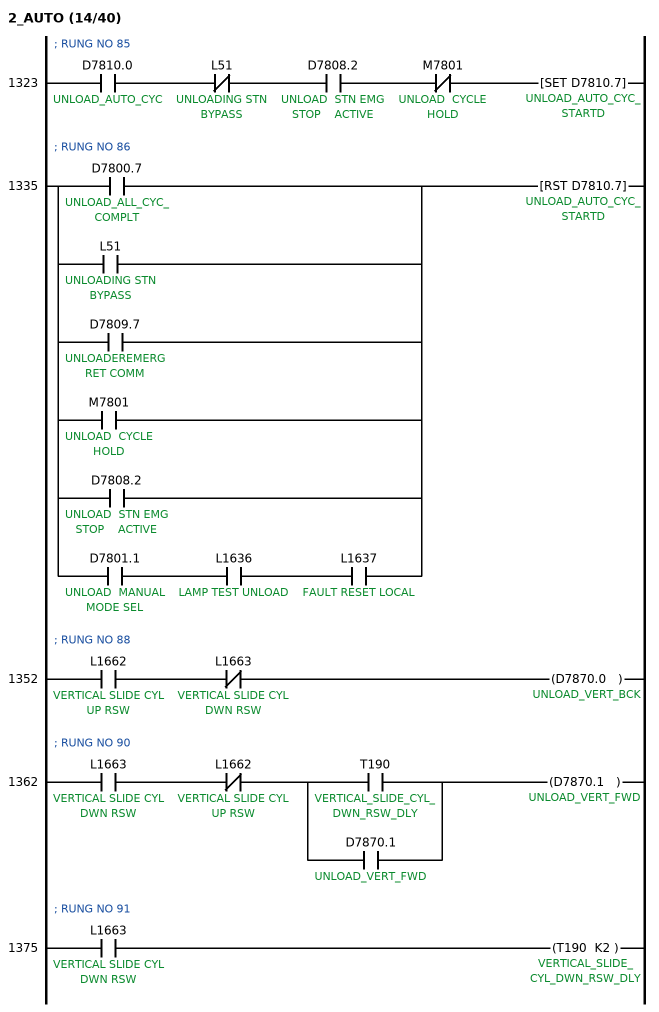
; RUNG NO 85
1323  LD      D7810.0  ; UNLOAD_AUTO_CYC
      ANI     L51  ; UNLOADING STN BYPASS
      AND     D7808.2  ; UNLOAD  STN EMG STOP    ACTIVE
      ANI     M7801  ; UNLOAD  CYCLE   HOLD
      SET     D7810.7  ; UNLOAD_AUTO_CYC_STARTD
; RUNG NO 86
1335  LD      D7800.7  ; UNLOAD_ALL_CYC_COMPLT
      OR      L51  ; UNLOADING STN BYPASS
      OR      D7809.7  ; UNLOADEREMERG   RET COMM
      OR      M7801  ; UNLOAD  CYCLE   HOLD
      OR      D7808.2  ; UNLOAD  STN EMG STOP    ACTIVE
      LD      D7801.1  ; UNLOAD  MANUAL  MODE SEL
      AND     L1636  ; LAMP TEST UNLOAD
      AND     L1637  ; FAULT RESET LOCAL
      ORB
      RST     D7810.7  ; UNLOAD_AUTO_CYC_STARTD
; RUNG NO 88
1352  LD      L1662  ; VERTICAL SLIDE CYL UP RSW
      ANI     L1663  ; VERTICAL SLIDE CYL DWN RSW
      OUT     D7870.0  ; UNLOAD_VERT_BCK
; RUNG NO 90
1362  LD      L1663  ; VERTICAL SLIDE CYL DWN RSW
      ANI     L1662  ; VERTICAL SLIDE CYL UP RSW
      LD      T190  ; VERTICAL_SLIDE_CYL_DWN_RSW_DLY
      OR      D7870.1  ; UNLOAD_VERT_FWD
      ANB
      OUT     D7870.1  ; UNLOAD_VERT_FWD
; RUNG NO 91
1375  LD      L1663  ; VERTICAL SLIDE CYL DWN RSW
      OUT     T190 K2  ; VERTICAL_SLIDE_CYL_DWN_RSW_DLY
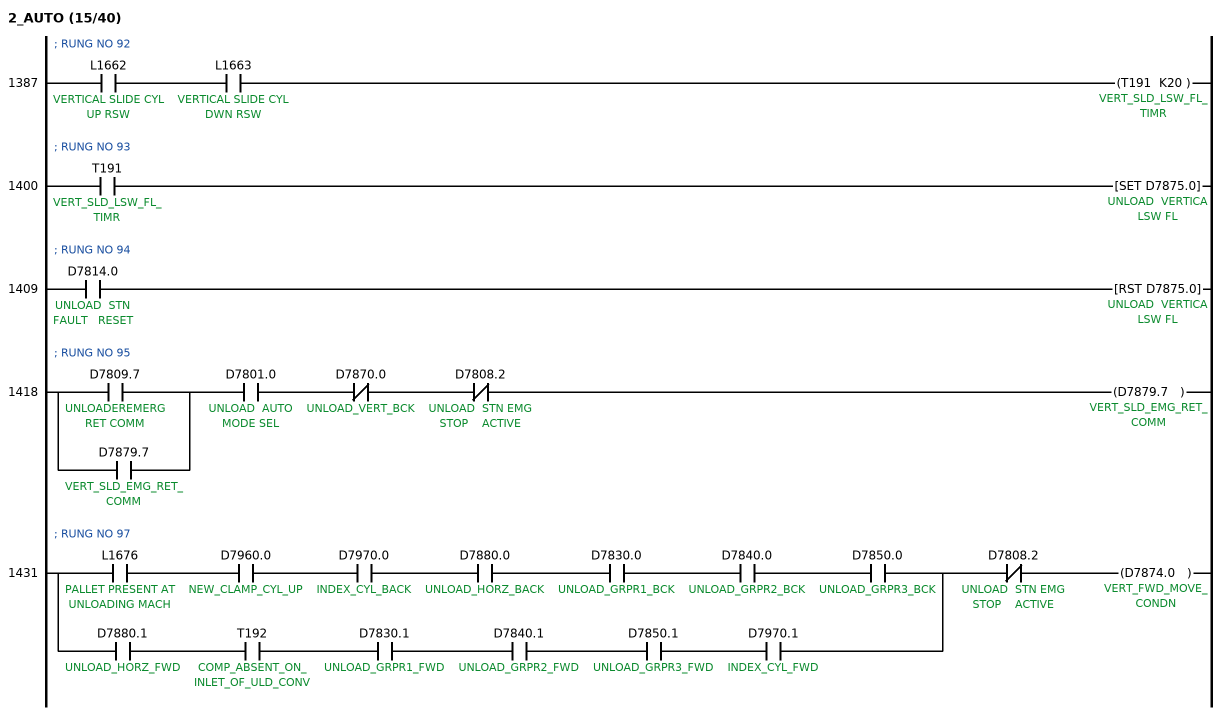
; RUNG NO 92
1387  LD      L1662  ; VERTICAL SLIDE CYL UP RSW
      AND     L1663  ; VERTICAL SLIDE CYL DWN RSW
      OUT     T191 K20  ; VERT_SLD_LSW_FL_TIMR
; RUNG NO 93
1400  LD      T191  ; VERT_SLD_LSW_FL_TIMR
      SET     D7875.0  ; UNLOAD  VERTICA LSW FL
; RUNG NO 94
1409  LD      D7814.0  ; UNLOAD  STN     FAULT   RESET
      RST     D7875.0  ; UNLOAD  VERTICA LSW FL
; RUNG NO 95
1418  LD      D7809.7  ; UNLOADEREMERG   RET COMM
      OR      D7879.7  ; VERT_SLD_EMG_RET_COMM
      AND     D7801.0  ; UNLOAD  AUTO    MODE SEL
      ANI     D7870.0  ; UNLOAD_VERT_BCK
      ANI     D7808.2  ; UNLOAD  STN EMG STOP    ACTIVE
      OUT     D7879.7  ; VERT_SLD_EMG_RET_COMM
; RUNG NO 97
1431  LD      L1676  ; PALLET PRESENT AT UNLOADING MACH
      AND     D7960.0  ; NEW_CLAMP_CYL_UP
      AND     D7970.0  ; INDEX_CYL_BACK
      AND     D7880.0  ; UNLOAD_HORZ_BACK
      AND     D7830.0  ; UNLOAD_GRPR1_BCK
      AND     D7840.0  ; UNLOAD_GRPR2_BCK
      AND     D7850.0  ; UNLOAD_GRPR3_BCK
      LD      D7880.1  ; UNLOAD_HORZ_FWD
      AND     T192  ; COMP_ABSENT_ON_INLET_OF_ULD_CONV
      AND     D7830.1  ; UNLOAD_GRPR1_FWD
      AND     D7840.1  ; UNLOAD_GRPR2_FWD
      AND     D7850.1  ; UNLOAD_GRPR3_FWD
      AND     D7970.1  ; INDEX_CYL_FWD
      ORB
      ANI     D7808.2  ; UNLOAD  STN EMG STOP    ACTIVE
      OUT     D7874.0  ; VERT_FWD_MOVE_CONDN
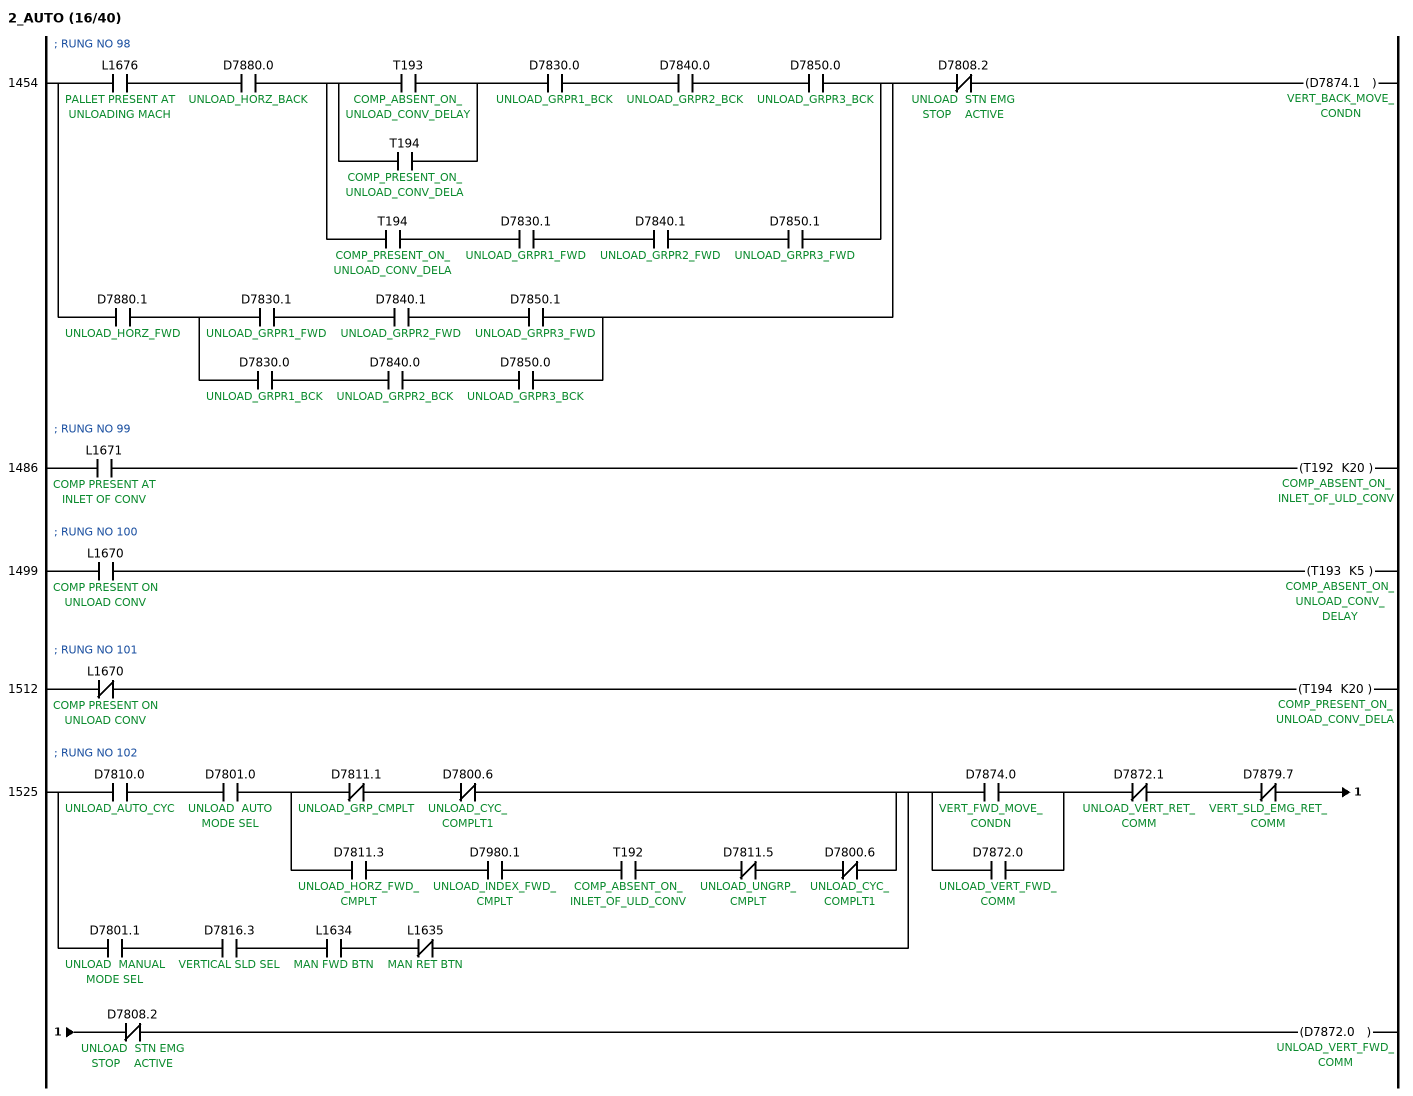
; RUNG NO 98
1454  LD      L1676  ; PALLET PRESENT AT UNLOADING MACH
      AND     D7880.0  ; UNLOAD_HORZ_BACK
      LD      T193  ; COMP_ABSENT_ON_UNLOAD_CONV_DELAY
      OR      T194  ; COMP_PRESENT_ON_UNLOAD_CONV_DELA
      AND     D7830.0  ; UNLOAD_GRPR1_BCK
      AND     D7840.0  ; UNLOAD_GRPR2_BCK
      AND     D7850.0  ; UNLOAD_GRPR3_BCK
      LD      T194  ; COMP_PRESENT_ON_UNLOAD_CONV_DELA
      AND     D7830.1  ; UNLOAD_GRPR1_FWD
      AND     D7840.1  ; UNLOAD_GRPR2_FWD
      AND     D7850.1  ; UNLOAD_GRPR3_FWD
      ORB
      ANB
      LD      D7880.1  ; UNLOAD_HORZ_FWD
      LD      D7830.1  ; UNLOAD_GRPR1_FWD
      AND     D7840.1  ; UNLOAD_GRPR2_FWD
      AND     D7850.1  ; UNLOAD_GRPR3_FWD
      LD      D7830.0  ; UNLOAD_GRPR1_BCK
      AND     D7840.0  ; UNLOAD_GRPR2_BCK
      AND     D7850.0  ; UNLOAD_GRPR3_BCK
      ORB
      ANB
      ORB
      ANI     D7808.2  ; UNLOAD  STN EMG STOP    ACTIVE
      OUT     D7874.1  ; VERT_BACK_MOVE_CONDN
; RUNG NO 99
1486  LD      L1671  ; COMP PRESENT AT INLET OF CONV
      OUT     T192 K20  ; COMP_ABSENT_ON_INLET_OF_ULD_CONV
; RUNG NO 100
1499  LD      L1670  ; COMP PRESENT ON UNLOAD CONV
      OUT     T193 K5  ; COMP_ABSENT_ON_UNLOAD_CONV_DELAY
; RUNG NO 101
1512  LDI     L1670  ; COMP PRESENT ON UNLOAD CONV
      OUT     T194 K20  ; COMP_PRESENT_ON_UNLOAD_CONV_DELA
; RUNG NO 102
1525  LD      D7810.0  ; UNLOAD_AUTO_CYC
      AND     D7801.0  ; UNLOAD  AUTO    MODE SEL
      LDI     D7811.1  ; UNLOAD_GRP_CMPLT
      ANI     D7800.6  ; UNLOAD_CYC_COMPLT1
      LD      D7811.3  ; UNLOAD_HORZ_FWD_CMPLT
      AND     D7980.1  ; UNLOAD_INDEX_FWD_CMPLT
      AND     T192  ; COMP_ABSENT_ON_INLET_OF_ULD_CONV
      ANI     D7811.5  ; UNLOAD_UNGRP_CMPLT
      ANI     D7800.6  ; UNLOAD_CYC_COMPLT1
      ORB
      ANB
      LD      D7801.1  ; UNLOAD  MANUAL  MODE SEL
      AND     D7816.3  ; VERTICAL SLD SEL
      AND     L1634  ; MAN FWD BTN
      ANI     L1635  ; MAN RET BTN
      ORB
      LD      D7874.0  ; VERT_FWD_MOVE_CONDN
      OR      D7872.0  ; UNLOAD_VERT_FWD_COMM
      ANB
      ANI     D7872.1  ; UNLOAD_VERT_RET_COMM
      ANI     D7879.7  ; VERT_SLD_EMG_RET_COMM
      ANI     D7808.2  ; UNLOAD  STN EMG STOP    ACTIVE
      OUT     D7872.0  ; UNLOAD_VERT_FWD_COMM
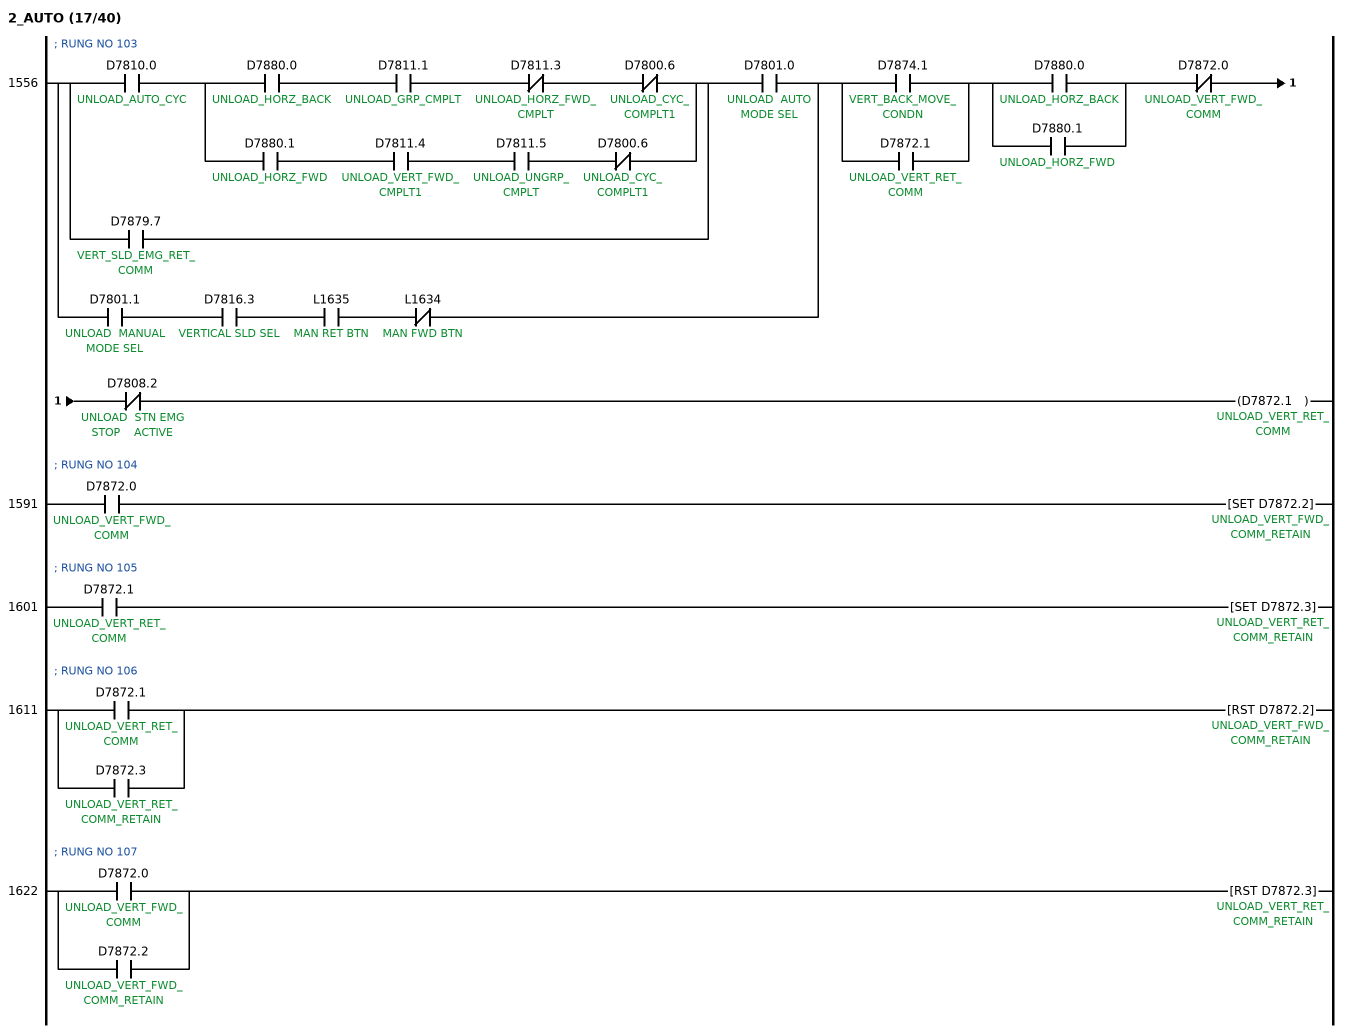
; RUNG NO 103
1556  LD      D7810.0  ; UNLOAD_AUTO_CYC
      LD      D7880.0  ; UNLOAD_HORZ_BACK
      AND     D7811.1  ; UNLOAD_GRP_CMPLT
      ANI     D7811.3  ; UNLOAD_HORZ_FWD_CMPLT
      ANI     D7800.6  ; UNLOAD_CYC_COMPLT1
      LD      D7880.1  ; UNLOAD_HORZ_FWD
      AND     D7811.4  ; UNLOAD_VERT_FWD_CMPLT1
      AND     D7811.5  ; UNLOAD_UNGRP_CMPLT
      ANI     D7800.6  ; UNLOAD_CYC_COMPLT1
      ORB
      ANB
      OR      D7879.7  ; VERT_SLD_EMG_RET_COMM
      AND     D7801.0  ; UNLOAD  AUTO    MODE SEL
      LD      D7801.1  ; UNLOAD  MANUAL  MODE SEL
      AND     D7816.3  ; VERTICAL SLD SEL
      AND     L1635  ; MAN RET BTN
      ANI     L1634  ; MAN FWD BTN
      ORB
      LD      D7874.1  ; VERT_BACK_MOVE_CONDN
      OR      D7872.1  ; UNLOAD_VERT_RET_COMM
      ANB
      LD      D7880.0  ; UNLOAD_HORZ_BACK
      OR      D7880.1  ; UNLOAD_HORZ_FWD
      ANB
      ANI     D7872.0  ; UNLOAD_VERT_FWD_COMM
      ANI     D7808.2  ; UNLOAD  STN EMG STOP    ACTIVE
      OUT     D7872.1  ; UNLOAD_VERT_RET_COMM
; RUNG NO 104
1591  LD      D7872.0  ; UNLOAD_VERT_FWD_COMM
      SET     D7872.2  ; UNLOAD_VERT_FWD_COMM_RETAIN
; RUNG NO 105
1601  LD      D7872.1  ; UNLOAD_VERT_RET_COMM
      SET     D7872.3  ; UNLOAD_VERT_RET_COMM_RETAIN
; RUNG NO 106
1611  LD      D7872.1  ; UNLOAD_VERT_RET_COMM
      OR      D7872.3  ; UNLOAD_VERT_RET_COMM_RETAIN
      RST     D7872.2  ; UNLOAD_VERT_FWD_COMM_RETAIN
; RUNG NO 107
1622  LD      D7872.0  ; UNLOAD_VERT_FWD_COMM
      OR      D7872.2  ; UNLOAD_VERT_FWD_COMM_RETAIN
      RST     D7872.3  ; UNLOAD_VERT_RET_COMM_RETAIN
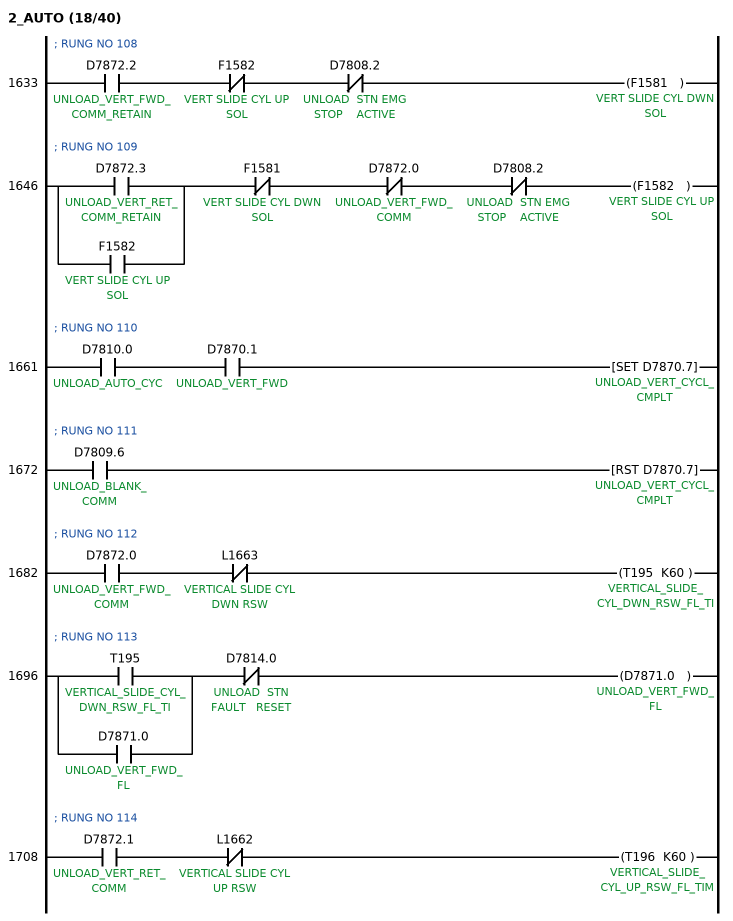
; RUNG NO 108
1633  LD      D7872.2  ; UNLOAD_VERT_FWD_COMM_RETAIN
      ANI     F1582  ; VERT SLIDE CYL UP SOL
      ANI     D7808.2  ; UNLOAD  STN EMG STOP    ACTIVE
      OUT     F1581  ; VERT SLIDE CYL DWN SOL
; RUNG NO 109
1646  LD      D7872.3  ; UNLOAD_VERT_RET_COMM_RETAIN
      OR      F1582  ; VERT SLIDE CYL UP SOL
      ANI     F1581  ; VERT SLIDE CYL DWN SOL
      ANI     D7872.0  ; UNLOAD_VERT_FWD_COMM
      ANI     D7808.2  ; UNLOAD  STN EMG STOP    ACTIVE
      OUT     F1582  ; VERT SLIDE CYL UP SOL
; RUNG NO 110
1661  LD      D7810.0  ; UNLOAD_AUTO_CYC
      AND     D7870.1  ; UNLOAD_VERT_FWD
      SET     D7870.7  ; UNLOAD_VERT_CYCL_CMPLT
; RUNG NO 111
1672  LD      D7809.6  ; UNLOAD_BLANK_COMM
      RST     D7870.7  ; UNLOAD_VERT_CYCL_CMPLT
; RUNG NO 112
1682  LD      D7872.0  ; UNLOAD_VERT_FWD_COMM
      ANI     L1663  ; VERTICAL SLIDE CYL DWN RSW
      OUT     T195 K60  ; VERTICAL_SLIDE_CYL_DWN_RSW_FL_TI
; RUNG NO 113
1696  LD      T195  ; VERTICAL_SLIDE_CYL_DWN_RSW_FL_TI
      OR      D7871.0  ; UNLOAD_VERT_FWD_FL
      ANI     D7814.0  ; UNLOAD  STN     FAULT   RESET
      OUT     D7871.0  ; UNLOAD_VERT_FWD_FL
; RUNG NO 114
1708  LD      D7872.1  ; UNLOAD_VERT_RET_COMM
      ANI     L1662  ; VERTICAL SLIDE CYL UP RSW
      OUT     T196 K60  ; VERTICAL_SLIDE_CYL_UP_RSW_FL_TIM
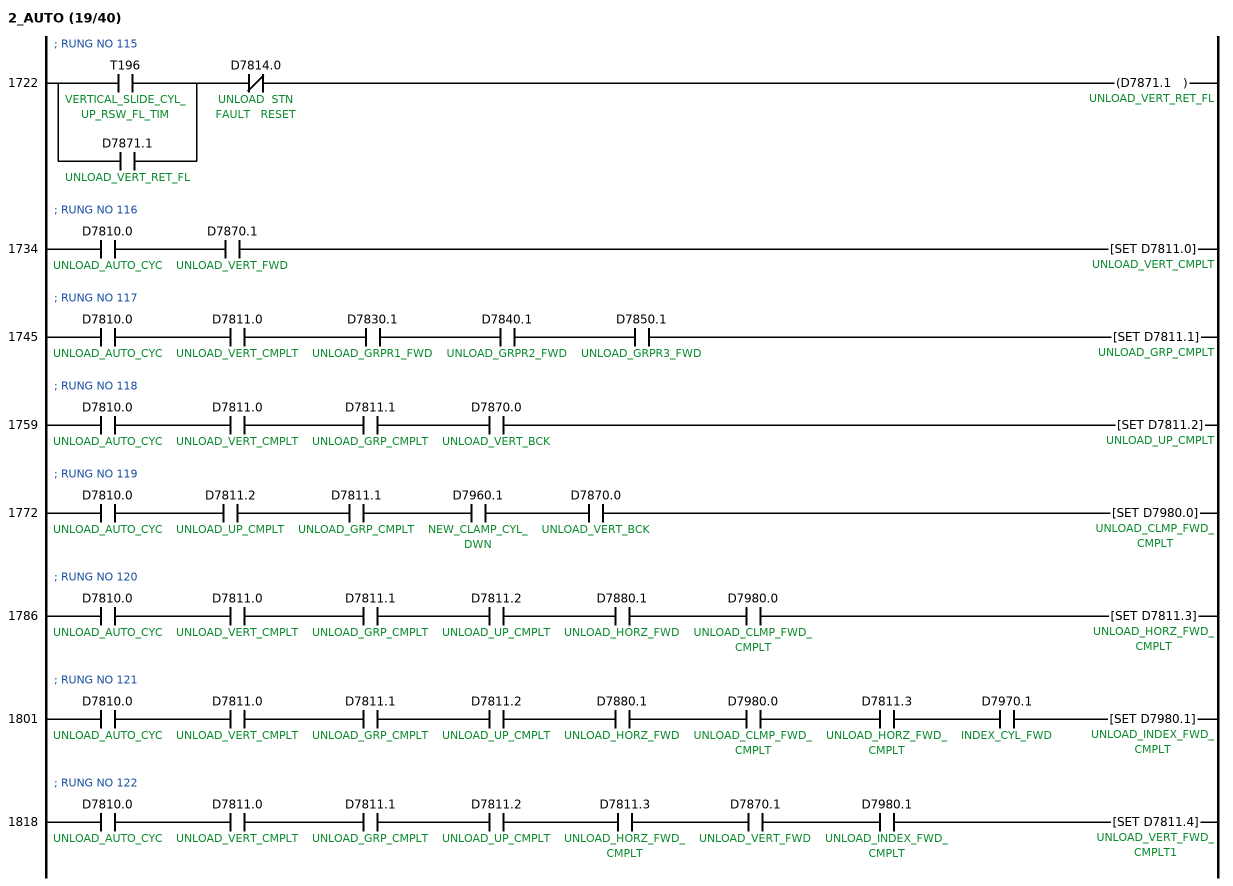
; RUNG NO 115
1722  LD      T196  ; VERTICAL_SLIDE_CYL_UP_RSW_FL_TIM
      OR      D7871.1  ; UNLOAD_VERT_RET_FL
      ANI     D7814.0  ; UNLOAD  STN     FAULT   RESET
      OUT     D7871.1  ; UNLOAD_VERT_RET_FL
; RUNG NO 116
1734  LD      D7810.0  ; UNLOAD_AUTO_CYC
      AND     D7870.1  ; UNLOAD_VERT_FWD
      SET     D7811.0  ; UNLOAD_VERT_CMPLT
; RUNG NO 117
1745  LD      D7810.0  ; UNLOAD_AUTO_CYC
      AND     D7811.0  ; UNLOAD_VERT_CMPLT
      AND     D7830.1  ; UNLOAD_GRPR1_FWD
      AND     D7840.1  ; UNLOAD_GRPR2_FWD
      AND     D7850.1  ; UNLOAD_GRPR3_FWD
      SET     D7811.1  ; UNLOAD_GRP_CMPLT
; RUNG NO 118
1759  LD      D7810.0  ; UNLOAD_AUTO_CYC
      AND     D7811.0  ; UNLOAD_VERT_CMPLT
      AND     D7811.1  ; UNLOAD_GRP_CMPLT
      AND     D7870.0  ; UNLOAD_VERT_BCK
      SET     D7811.2  ; UNLOAD_UP_CMPLT
; RUNG NO 119
1772  LD      D7810.0  ; UNLOAD_AUTO_CYC
      AND     D7811.2  ; UNLOAD_UP_CMPLT
      AND     D7811.1  ; UNLOAD_GRP_CMPLT
      AND     D7960.1  ; NEW_CLAMP_CYL_DWN
      AND     D7870.0  ; UNLOAD_VERT_BCK
      SET     D7980.0  ; UNLOAD_CLMP_FWD_CMPLT
; RUNG NO 120
1786  LD      D7810.0  ; UNLOAD_AUTO_CYC
      AND     D7811.0  ; UNLOAD_VERT_CMPLT
      AND     D7811.1  ; UNLOAD_GRP_CMPLT
      AND     D7811.2  ; UNLOAD_UP_CMPLT
      AND     D7880.1  ; UNLOAD_HORZ_FWD
      AND     D7980.0  ; UNLOAD_CLMP_FWD_CMPLT
      SET     D7811.3  ; UNLOAD_HORZ_FWD_CMPLT
; RUNG NO 121
1801  LD      D7810.0  ; UNLOAD_AUTO_CYC
      AND     D7811.0  ; UNLOAD_VERT_CMPLT
      AND     D7811.1  ; UNLOAD_GRP_CMPLT
      AND     D7811.2  ; UNLOAD_UP_CMPLT
      AND     D7880.1  ; UNLOAD_HORZ_FWD
      AND     D7980.0  ; UNLOAD_CLMP_FWD_CMPLT
      AND     D7811.3  ; UNLOAD_HORZ_FWD_CMPLT
      AND     D7970.1  ; INDEX_CYL_FWD
      SET     D7980.1  ; UNLOAD_INDEX_FWD_CMPLT
; RUNG NO 122
1818  LD      D7810.0  ; UNLOAD_AUTO_CYC
      AND     D7811.0  ; UNLOAD_VERT_CMPLT
      AND     D7811.1  ; UNLOAD_GRP_CMPLT
      AND     D7811.2  ; UNLOAD_UP_CMPLT
      AND     D7811.3  ; UNLOAD_HORZ_FWD_CMPLT
      AND     D7870.1  ; UNLOAD_VERT_FWD
      AND     D7980.1  ; UNLOAD_INDEX_FWD_CMPLT
      SET     D7811.4  ; UNLOAD_VERT_FWD_CMPLT1
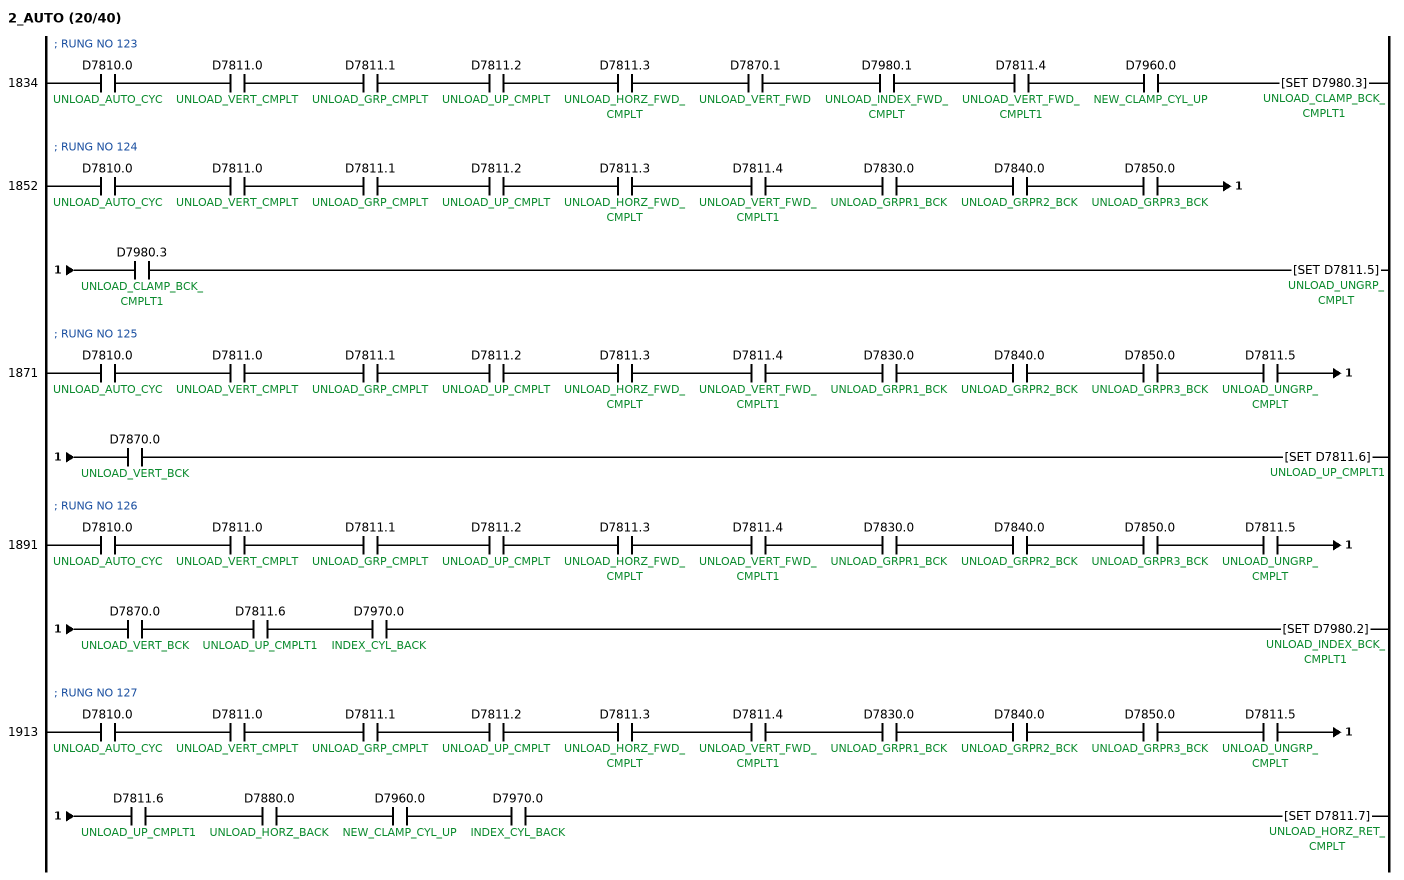
; RUNG NO 123
1834  LD      D7810.0  ; UNLOAD_AUTO_CYC
      AND     D7811.0  ; UNLOAD_VERT_CMPLT
      AND     D7811.1  ; UNLOAD_GRP_CMPLT
      AND     D7811.2  ; UNLOAD_UP_CMPLT
      AND     D7811.3  ; UNLOAD_HORZ_FWD_CMPLT
      AND     D7870.1  ; UNLOAD_VERT_FWD
      AND     D7980.1  ; UNLOAD_INDEX_FWD_CMPLT
      AND     D7811.4  ; UNLOAD_VERT_FWD_CMPLT1
      AND     D7960.0  ; NEW_CLAMP_CYL_UP
      SET     D7980.3  ; UNLOAD_CLAMP_BCK_CMPLT1
; RUNG NO 124
1852  LD      D7810.0  ; UNLOAD_AUTO_CYC
      AND     D7811.0  ; UNLOAD_VERT_CMPLT
      AND     D7811.1  ; UNLOAD_GRP_CMPLT
      AND     D7811.2  ; UNLOAD_UP_CMPLT
      AND     D7811.3  ; UNLOAD_HORZ_FWD_CMPLT
      AND     D7811.4  ; UNLOAD_VERT_FWD_CMPLT1
      AND     D7830.0  ; UNLOAD_GRPR1_BCK
      AND     D7840.0  ; UNLOAD_GRPR2_BCK
      AND     D7850.0  ; UNLOAD_GRPR3_BCK
      AND     D7980.3  ; UNLOAD_CLAMP_BCK_CMPLT1
      SET     D7811.5  ; UNLOAD_UNGRP_CMPLT
; RUNG NO 125
1871  LD      D7810.0  ; UNLOAD_AUTO_CYC
      AND     D7811.0  ; UNLOAD_VERT_CMPLT
      AND     D7811.1  ; UNLOAD_GRP_CMPLT
      AND     D7811.2  ; UNLOAD_UP_CMPLT
      AND     D7811.3  ; UNLOAD_HORZ_FWD_CMPLT
      AND     D7811.4  ; UNLOAD_VERT_FWD_CMPLT1
      AND     D7830.0  ; UNLOAD_GRPR1_BCK
      AND     D7840.0  ; UNLOAD_GRPR2_BCK
      AND     D7850.0  ; UNLOAD_GRPR3_BCK
      AND     D7811.5  ; UNLOAD_UNGRP_CMPLT
      AND     D7870.0  ; UNLOAD_VERT_BCK
      SET     D7811.6  ; UNLOAD_UP_CMPLT1
; RUNG NO 126
1891  LD      D7810.0  ; UNLOAD_AUTO_CYC
      AND     D7811.0  ; UNLOAD_VERT_CMPLT
      AND     D7811.1  ; UNLOAD_GRP_CMPLT
      AND     D7811.2  ; UNLOAD_UP_CMPLT
      AND     D7811.3  ; UNLOAD_HORZ_FWD_CMPLT
      AND     D7811.4  ; UNLOAD_VERT_FWD_CMPLT1
      AND     D7830.0  ; UNLOAD_GRPR1_BCK
      AND     D7840.0  ; UNLOAD_GRPR2_BCK
      AND     D7850.0  ; UNLOAD_GRPR3_BCK
      AND     D7811.5  ; UNLOAD_UNGRP_CMPLT
      AND     D7870.0  ; UNLOAD_VERT_BCK
      AND     D7811.6  ; UNLOAD_UP_CMPLT1
      AND     D7970.0  ; INDEX_CYL_BACK
      SET     D7980.2  ; UNLOAD_INDEX_BCK_CMPLT1
; RUNG NO 127
1913  LD      D7810.0  ; UNLOAD_AUTO_CYC
      AND     D7811.0  ; UNLOAD_VERT_CMPLT
      AND     D7811.1  ; UNLOAD_GRP_CMPLT
      AND     D7811.2  ; UNLOAD_UP_CMPLT
      AND     D7811.3  ; UNLOAD_HORZ_FWD_CMPLT
      AND     D7811.4  ; UNLOAD_VERT_FWD_CMPLT1
      AND     D7830.0  ; UNLOAD_GRPR1_BCK
      AND     D7840.0  ; UNLOAD_GRPR2_BCK
      AND     D7850.0  ; UNLOAD_GRPR3_BCK
      AND     D7811.5  ; UNLOAD_UNGRP_CMPLT
      AND     D7811.6  ; UNLOAD_UP_CMPLT1
      AND     D7880.0  ; UNLOAD_HORZ_BACK
      AND     D7960.0  ; NEW_CLAMP_CYL_UP
      AND     D7970.0  ; INDEX_CYL_BACK
      SET     D7811.7  ; UNLOAD_HORZ_RET_CMPLT
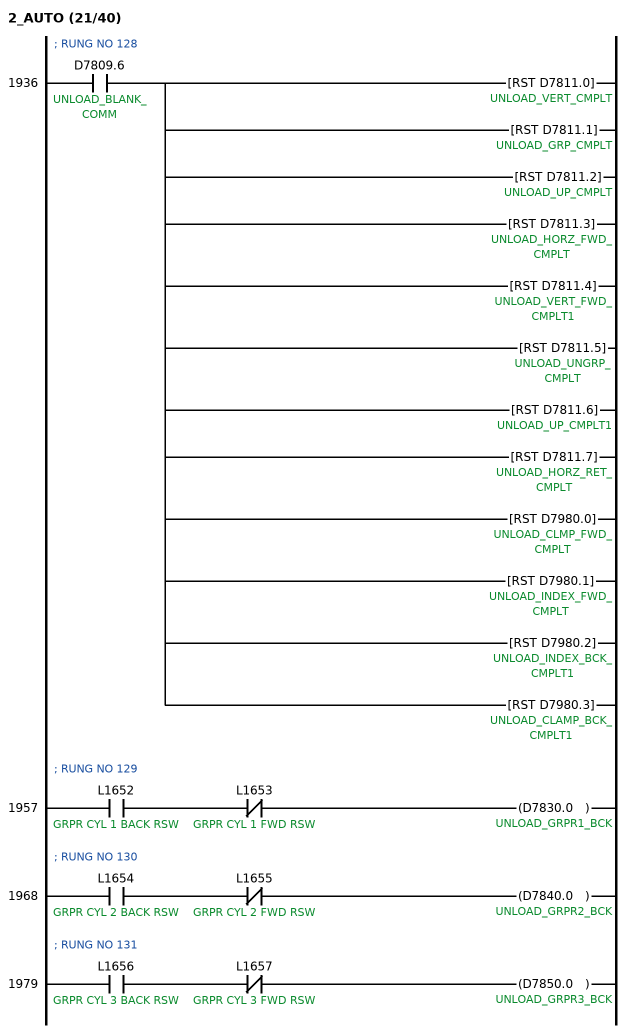
; RUNG NO 128
1936  LD      D7809.6  ; UNLOAD_BLANK_COMM
      RST     D7811.0  ; UNLOAD_VERT_CMPLT
      RST     D7811.1  ; UNLOAD_GRP_CMPLT
      RST     D7811.2  ; UNLOAD_UP_CMPLT
      RST     D7811.3  ; UNLOAD_HORZ_FWD_CMPLT
      RST     D7811.4  ; UNLOAD_VERT_FWD_CMPLT1
      RST     D7811.5  ; UNLOAD_UNGRP_CMPLT
      RST     D7811.6  ; UNLOAD_UP_CMPLT1
      RST     D7811.7  ; UNLOAD_HORZ_RET_CMPLT
      RST     D7980.0  ; UNLOAD_CLMP_FWD_CMPLT
      RST     D7980.1  ; UNLOAD_INDEX_FWD_CMPLT
      RST     D7980.2  ; UNLOAD_INDEX_BCK_CMPLT1
      RST     D7980.3  ; UNLOAD_CLAMP_BCK_CMPLT1
; RUNG NO 129
1957  LD      L1652  ; GRPR CYL 1 BACK RSW
      ANI     L1653  ; GRPR CYL 1 FWD RSW
      OUT     D7830.0  ; UNLOAD_GRPR1_BCK
; RUNG NO 130
1968  LD      L1654  ; GRPR CYL 2 BACK RSW
      ANI     L1655  ; GRPR CYL 2 FWD RSW
      OUT     D7840.0  ; UNLOAD_GRPR2_BCK
; RUNG NO 131
1979  LD      L1656  ; GRPR CYL 3 BACK RSW
      ANI     L1657  ; GRPR CYL 3 FWD RSW
      OUT     D7850.0  ; UNLOAD_GRPR3_BCK
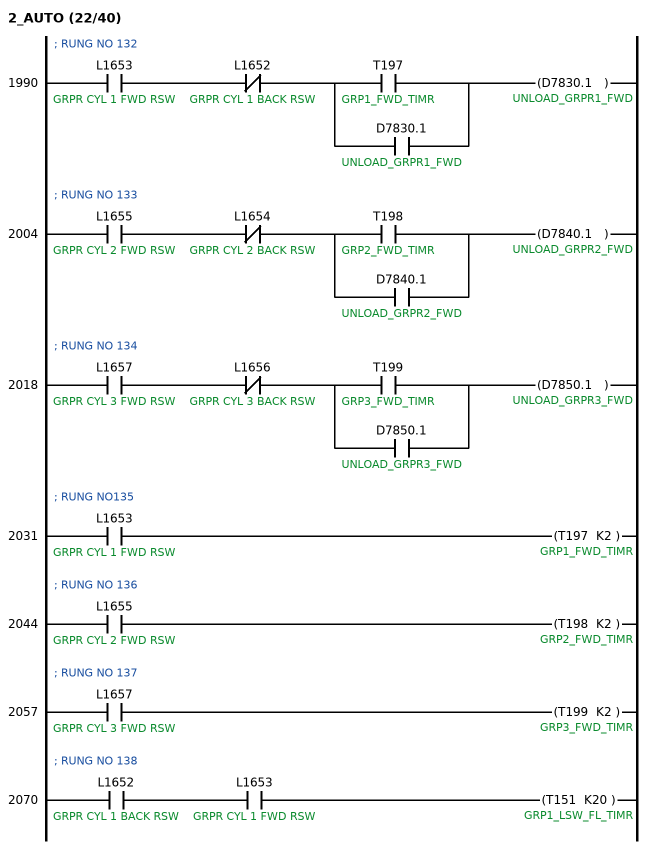
; RUNG NO 132
1990  LD      L1653  ; GRPR CYL 1 FWD RSW
      ANI     L1652  ; GRPR CYL 1 BACK RSW
      LD      T197  ; GRP1_FWD_TIMR
      OR      D7830.1  ; UNLOAD_GRPR1_FWD
      ANB
      OUT     D7830.1  ; UNLOAD_GRPR1_FWD
; RUNG NO 133
2004  LD      L1655  ; GRPR CYL 2 FWD RSW
      ANI     L1654  ; GRPR CYL 2 BACK RSW
      LD      T198  ; GRP2_FWD_TIMR
      OR      D7840.1  ; UNLOAD_GRPR2_FWD
      ANB
      OUT     D7840.1  ; UNLOAD_GRPR2_FWD
; RUNG NO 134
2018  LD      L1657  ; GRPR CYL 3 FWD RSW
      ANI     L1656  ; GRPR CYL 3 BACK RSW
      LD      T199  ; GRP3_FWD_TIMR
      OR      D7850.1  ; UNLOAD_GRPR3_FWD
      ANB
      OUT     D7850.1  ; UNLOAD_GRPR3_FWD
; RUNG NO135
2031  LD      L1653  ; GRPR CYL 1 FWD RSW
      OUT     T197 K2  ; GRP1_FWD_TIMR
; RUNG NO 136
2044  LD      L1655  ; GRPR CYL 2 FWD RSW
      OUT     T198 K2  ; GRP2_FWD_TIMR
; RUNG NO 137
2057  LD      L1657  ; GRPR CYL 3 FWD RSW
      OUT     T199 K2  ; GRP3_FWD_TIMR
; RUNG NO 138
2070  LD      L1652  ; GRPR CYL 1 BACK RSW
      AND     L1653  ; GRPR CYL 1 FWD RSW
      OUT     T151 K20  ; GRP1_LSW_FL_TIMR
